# B&R Automation Studio project Nitto (part 13)

#### FB_Machine.st - TODO: Beinhaltet aller Baugrupen der Maschine
```iecst
(********************************************************************
 * COPYRIGHT -- Microsoft
 ********************************************************************
 * Library: UserSpilke
 * Datei: FB_Machine.st
 * Autor: Awalz
 * Erstellt: 24. März 2014
 ********************************************************************
 * Implementierung der Library UserSpilke
 ********************************************************************)

(* TODO: Beinhaltet aller Baugrupen der Maschine *)
FUNCTION_BLOCK FB_Machine

	ctrl(masterModul := masterModul,
		UnwinderUnit := UnwinderUnit,
		webbuffer := webbuffer,
		pullbreak := pullbreak ,
		cuttingunit1 := cuttingunit1,
		turngridwinder := turngridwinder,
		longcutter := longcutter,
		pullbreakSt := pullbreakSt,
		cuttingunit2 :=	cuttingunit2,
		catchbelt := catchbelt,
		conveyor := conveyor,
		webguidingbuffer := webguidingbuffer,
		webguiding := webguiding,
		emcy_inputs := emcy_inputs,summerystartstop := summerystartstop,
		IOs := IOs, panel := panel, safety := safety, gVarMachine := gVarMachine, switchcabinet := switchcabinet,
		packbelt := packbelt);  (**)

END_FUNCTION_BLOCK
```

#### FB_MachineIOs.st
```iecst
(********************************************************************
 * COPYRIGHT -- Microsoft
 ********************************************************************
 * Programm: MAIN
 * Datei: FB_MachineIOs.st
 * Autor: Awalz
 * Erstellt: 12. Mai 2014
 ********************************************************************
 * Implementierung des Programms MAIN
 ********************************************************************)

 (*<$Description$> TODO: Bitte Kommentar hier einzufügen </$Description$>*)
FUNCTION_BLOCK FB_MachineIOs
	ampel(clk := panel.clk);
	CEEPlug_o := CEEPlugON;
END_FUNCTION_BLOCK
```

#### Package Logical/MainMachineCtrl/MAIN/Mastermodul - Neues leeres Paket

#### FB_SpeedCtlrPid.st
```iecst
(********************************************************************
 * COPYRIGHT -- Microsoft
 ********************************************************************
 * Programm: MAIN
 * Datei: FB_SpeedCtlrPid.st
 * Autor: awalz
 * Erstellt: 10. Dezember 2014
 ********************************************************************
 * Implementierung des Programms MAIN
 ********************************************************************)

(* TODO: Bitte Kommentar hier einfügen *)
FUNCTION_BLOCK FB_SpeedCtlrPid
	IF firststart THEN
		LCRPIDpara_0.Kfbk			:= 2.0; // Anti-windup used
		LCRPIDpara_0.d_mode			:= LCRPID_D_MODE_E;	// differentiate control deviation
		LCRPIDpara_0.fbk_mode		:= LCRPID_FBK_MODE_INTERN;	// feedback of internal output
		LCRPID_0.mode				:= LCRPID_MODE_AUTO;	// Standard PID operating mod
		// 50.000 = 3 m/min
		LCRPID_0.Y_max				:= 10;	// percent
		LCRPID_0.Y_min				:= -10;// percent
		LCRPIDpara_0.invert			:= TRUE;
		LCRPIDpara_0.Kp				:= PID_Kp; //1.6; (*11*)//0.2//17.09.15 geändert
		LCRPIDpara_0.Tn				:= 7;// 6;	//(*1.1*)//7 //17.09.15 geändert
		LCRPIDpara_0.Tv				:= 0.0; // D-part
		LCRPIDpara_0.Tf				:= 0;(*0.020;*)
		LCRPIDpara_0.WX_max			:= 1000.0;
		LCRPIDpara_0.WX_min			:= -1000.0;
		LCRPID_0.ident				:= LCRPIDpara_0.ident;
		zeitkonstante				:= 0.1;
		lowPassEnable				:= TRUE;
		// Maximum controller output:
		firststart := FALSE;
	 END_IF
	lowPass.enable := lowPassEnable;
	IF dancepos >32767 THEN (* weil der Sensor zu nahe sitzt gibt es ein Ünerlauf*)
		test := 2000;
	ELSE
		test := dancepos;
	END_IF
	lowPass.x := INT_TO_REAL (test);
	lowPass.t := zeitkonstante; //2
	lowPass();
	lowPassSpeed.enable := TRUE;
	lowPassSpeed.x := INT_TO_REAL (ConveyerVelocity); // analog Input from conveyer
	lowPassSpeed.t := 3;
	lowPassSpeed();
//	lowPass.y_set := 0;
//	lowPass.set := TRUE;
//	rDancepos := INT_TO_REAL (dancepos) * SCALE_10V_TO_MM;
	rDancepos := lowPass.y * SCALE_10V_TO_MM; // gefilterte Tänzer position in mm
	inc_to_volt := lowPassSpeed.y * SCALE_INC_TO_V;
	volt_to_speed := maxMainVelocity /10 * inc_to_volt;

	LCRPIDpara_0();
	//************************** LCRPID *******************************
	LCRPID_0.ident						:= LCRPIDpara_0.ident;
	// PID controller:
	//  setpoint  		"W" = dancer position from application recipe
	//  actual value	"X" = measured act dancer position from analog input (*override wird beim füllen draufgegebe*)
	LCRPID_0.W			:= LIMIT (0, setDancerpos , 1000);
	LCRPID_0.X			:= rDancepos;  (*LCRPT1e_ActTension.y;*)
	LCRPID_0();
	(*OutPID				:= LCRPID_TM.Y * TM_SCALE_PID_OUT_TO_OFFSET;*)

	IF reset THEN
		setVelocity := LIMIT (0, volt_to_speed, 21); (*setVelocity;*) (*+ velocityOffset;*) (* Offset damit der Tänzer in der Mitte bleibt*) // OKrebs // statt 11 -> 21
	ELSE
		IF lowPassSpeed.y < 600 THEN //  weil das Signal drunter nur ein Rauschen ist
			tempvalue	:= 0;
		ELSE
			tempvalue		:= LIMIT (-3, LCRPID_0.Y * TM_SCALE_PID_OUT_TO_OFFSET, 3(*maxMainVelocity*)) ;
		END_IF
//		setVelocity := LIMIT (0,( volt_to_speed + tempvalue), 11); // OKrebs 12.04.17

		IF startCycleWebturrit THEN  // OKrebs // 12.04.17 // ANFANG
			IF NOT dancerWasEmpty THEN (*1*)
				setVelocity := LIMIT (0, volt_to_speed + 2, 21); // Geschwindigkeit erhöhen bis Tänzer leer ist // // OKrebs // statt 11 -> 21
			END_IF
			IF rDancepos < minDancerPos THEN  (*2*)// Wenn Tänzer leer/oben ist
				setVelocity := LIMIT (0, speedToCycleWebturrit, 21); // Geschwindigkeit verringern bis der Tänzer wieder voll ist // // OKrebs // statt 11 -> 21
				dancerWasEmpty := TRUE;
			END_IF
			IF dancerWasEmpty AND (rDancepos > maxDancerPos) THEN (*3*) // Wenn Tänzer wieder voll ist
				startCycleWebturrit := FALSE;
			END_IF
		ELSE
			setVelocity := LIMIT (0,( volt_to_speed + tempvalue), 21);  // // OKrebs // statt 11 -> 21
			dancerWasEmpty := FALSE;
		END_IF // OKrebs // ENDE

	END_IF
	// ================
	// CHECK ERRORS
	// ================

	IF (LCRPID_0.status > 12022) AND
	   (LCRPID_0.status < 65534) THEN
//		// Error in PID controller detected -> stop control
		AxisStep		:= ST_CTRL_OFF;
	END_IF

	CASE AxisStep OF
		//********************* INITIALISATION ************************
		ST_INIT1:
			LCRPIDpara_0.enable		:= TRUE;
			LCRPIDpara_0.enter		:= FALSE;
			LCRPID_0.enable			:= FALSE; (* 10.12.14*)
			AxisStep					:= ST_READY;

		//********************* WAIT FOR COMMANDS ************************
		ST_READY:
				LCRPID_0.enable			:= FALSE;
				AxisStep		:= ST_WAIT_POWER_ENABLED;
			// End of STEP_TM_READY
		//********************* WAIT FOR DRIVES BEING ENABLED ************************
		ST_WAIT_POWER_ENABLED:
		(*	IF  MC_ReadStatus_0.StandStill OR  MC_ReadStatus_0.ContinuousMotion THEN*)
				AxisStep			:= ST_LOAD_PARA_START;
				// Generate rising edge at the enter input in order to update
				// PID controller parameters
				LCRPIDpara_0.enter	:= FALSE;
			// End of STEP_TM_WAIT_POWER_ENABLED
		//********************* START PARAMETER LOADING ************************
		ST_LOAD_PARA_START:
			// Rising edge for updating controller parameter
			LCRPIDpara_0.enter		:= TRUE;
			AxisStep				:= ST_WAIT_LOAD_PARA_DONE;
//		//********************* WAIT FOR PARAMETER LOAD COMPLETE ************************
		ST_WAIT_LOAD_PARA_DONE:
			LCRPIDpara_0.enter		:= FALSE;
			AxisStep				:= ST_WAIT_SWITCH_CTRL_ON;
			// End of STEP_TM_WAIT_LOAD_PARA_DONE
//
//		//********************* ACTIVATE CONTROL ************************
		ST_WAIT_SWITCH_CTRL_ON:
			IF   (LCRPIDpara_0.ident <> 0)  THEN
				// Enable PID controller and Offset correction for web tension control
				LCRPID_0.enable				:= TRUE;
			(*	AxisStep						:= ST_CTRL_ACTIVE*);
			ELSIF reset THEN
				AxisStep := ST_INIT1;
			END_IF

	END_CASE

END_FUNCTION_BLOCK
```

#### FB_MASTERMODUL.st
```iecst
(********************************************************************
 * COPYRIGHT -- Microsoft
 ********************************************************************
 * Library: UserSpilke
 * Datei: FB_MASTERMODUL.st
 * Autor: Awalz
 * Erstellt: 25. März 2014
 ********************************************************************
 * Implementierung der Library UserSpilke
 ********************************************************************)

(*<$Description$> TODO: Bitte Kommentar hier einzufügen </$Description$>*)
FUNCTION_BLOCK FB_MASTERMODUL
END_FUNCTION_BLOCK
```

#### ac_automaticMaster.st
```iecst
(********************************************************************
 * COPYRIGHT -- Microsoft
 ********************************************************************
 * Programm: MAIN
 * Datei: ac_automaticMaster.st
 * Autor: Awalz
 * Erstellt: 1. April 2014
 ********************************************************************
 * Implementierung des Programms MAIN
 ********************************************************************)

 (*<$Description$> Fügt eine neue Aktion zum IEC Programm oder Bibliothek </$Description$>*)
ACTION ac_automaticMaster:
	CASE state OF
	ST_IDLE:
	(*	pulsHorn(IN := FALSE);*)

		IF BetrCtrl.value = CONST.MACHINEMODES.AUTOMATIC THEN
			handWheel.reset := TRUE;
			panel.LDTAutomatic.LDT.aktion := CONST.LAMP.BLINK500;
			panel.LDTJOG.LDT.aktion := CONST.LAMP.OFF;
		(*	errorKlemmungVornUnten.active := FALSE;
			errorKlemmungHintenUnten.active := FALSE;
			IF unitsStatus.durchmesserStop THEN
				errorDiameterStop.active := TRUE;
			ELSE
				errorDiameterStop.active := FALSE;
				IF unitsStatus.klemmungVornStop THEN
					errorKlemmungVornUnten.active := TRUE;
				ELSIF unitsStatus.klemmungHintenStop THEN
					errorKlemmungHintenUnten.active := TRUE;
				ELSIF unitsStatus.unwinderNotUp THEN
					errorUnwinderNotUp.active := TRUE;
				ELSE
					errorUnwinderNotUp.active := FALSE;*)
					IF unitsStatus.ready AND cuttingunit2.emcy_inputs.EMCY_DoorsClosed AND  cuttingunit1.emcy_inputs.EMCY_DoorsClosed AND  webbuffer.emcy_inputs.EMCY_DoorsClosed AND pullbreak.emcy_inputs.EMCY_DoorsClosed AND
				 longcutter.emcy_inputs.EMCY_DoorsClosed AND cuttingunit2.emcy_inputs.EMCY_DoorsClosed  AND safety.RequestSLS THEN
					(*AND unitsStatus.clampingback AND unitsStatus.clampingfront AND unitsStatus.clampingsplicetable *)
						(*NOT (UnwinderUnit.clamp.toDown_o OR UnwinderUnit.splicetable.clampAfter.toDown_o OR
						UnwinderUnit.splicetable.clampBefore.toDown_o OR UnwinderUnit.unwinderDrv.clamp.toDown_o
						OR UnwinderUnit.unwinderOp.clamp.toDown_o) THEN*)
						(*AND datacom.mach.loaded AND datacom.recipe.loaded AND datacom.tools.com.loaded THEN*)
						state := ST_AXIS_RUN;
					END_IF
				(*END_IF
			END_IF*)
		ELSE
			err(reset := TRUE);
			busy := TRUE;
			StateCtrl := CTRL_AUTO_AFTER;
		END_IF

	ST_AXIS_RUN:
		IF axis.busy OR axis.cmd <> CONST.AXIS.NOACTION THEN
			axis.cmd := CONST.AXIS.NOACTION;
		ELSE
			panel.LDTAutomatic.LDT.aktion := CONST.LAMP.ON;
			IOs.ampel.ondelay := T#3s;
			IOs.ampel.horn := TRUE;
			axis(cmd := CONST.AXIS.MOVE_VELOCITY, velocity := handWheel.setVelocity);
			state := ST_AXIS_RUN_FAST;
		END_IF
	(*	ELSE
			data.set.override := 0;
			axis.ctrl.ref.PlcToNc.Override := data.set.override;
			axis.ctrl( cmd := CONST.AXIS.START, position := axis.ctrl.ref.NcToPlc.ActPos + 9999999999999, velocity := STARTVELO);
			panels.autoLangsam.lamp.aktion :=  const.LAMP.BLINK500;
			panels.autoSchnell.lamp.aktion :=  const.LAMP.BLINK500;

			IOs.tasterflascheAbwickler.jog.lamp.aktion := const.LAMP.BLINK500;
			IOs.tasterflascheLongford.jog.lamp.aktion := const.LAMP.BLINK500;
			IOs.tasterflscheSpender.jog.lamp.aktion := const.LAMP.BLINK500;
			state := ST_AXIS_RUN_FAST;
		END_IF*)

	ST_AXIS_RUN_FAST:
		axis();
		IF  NOT safety.RequestSLS THEN
			IOs.ampel.Gelb.aktion := CONST.LAMP.BLINK500;
			panel.LDTRESET.LDT.aktion := CONST.LAMP.BLINK500; (* um zu signalisieren dass der Safetyrequest gedückt werden muss*)
		ELSE
			IOs.ampel.Gelb.aktion := CONST.LAMP.OFF;
			panel.LDTRESET.LDT.aktion := CONST.LAMP.OFF;
		END_IF
		 // Geschwindigkeitsänderung mit Handrad auf dem Panel
		axis(cmd := CONST.AXIS.MOVE_VELOCITY, velocity := handWheel.setVelocity);
		IF BetrCtrl.value = CONST.MACHINEMODES.MANUAL THEN
//			errorKlemmungVornUnten.active := FALSE;
//			errorKlemmungHintenUnten.active := FALSE;
//			errorDiameterStop.active := FALSE;
//			errorUnwinderNotUp.active := FALSE;
			axis(cmd := CONST.AXIS.STOP, ruck := 0, verzoegerung := 120000 );
			state := ST_AXIS_STOP;
		ELSIF BetrCtrl.value <> CONST.MACHINEMODES.AUTOMATIC OR NOT unitsStatus.ready OR NOT safety.RequestSLS  THEN
//			errorKlemmungVornUnten.active := FALSE;
//			errorKlemmungHintenUnten.active := FALSE;
//			errorDiameterStop.active := FALSE;
//			errorUnwinderNotUp.active := FALSE;
			axis( cmd := CONST.AXIS.STOP, ruck := 20000, verzoegerung := 120000 );
			state := ST_AXIS_STOP;
		ELSIF unitsStatus.diameterStop THEN
//		(*errorKlemmungVornUnten.active := FALSE;
//			errorKlemmungHintenUnten.active := FALSE;
//			errorUnwinderNotUp.active := FALSE;
//			errorDiameterStop.active := TRUE;*)
			axis( cmd := CONST.AXIS.STOP, ruck := 20000, verzoegerung := 120000);
			state := ST_AXIS_STOP;
//		ELSIF 	unitsStatus.clampingfront THEN
//			(*errorKlemmungVornUnten.active := TRUE;
//			errorKlemmungHintenUnten.active := FALSE;
//			errorUnwinderNotUp.active := FALSE;
//			errorDiameterStop.active := FALSE;*)
//			axis( cmd := CONST.AXIS.STOP, ruck := 20000, verzoegerung := 4000 );
//		(*	panels.stopSchnell.lamp.aktion := const.LAMP.ON; (*J.H.*)
//			state := ST_AXIS_STOP;
//		ELSIF unitsStatus.clampingback THEN
//		(*	errorKlemmungVornUnten.active := FALSE;
//			errorKlemmungHintenUnten.active := TRUE;
//			errorUnwinderNotUp.active := FALSE;
//			errorDiameterStop.active := FALSE;*)
//			axis( cmd := CONST.AXIS.STOP, ruck := 20000, verzoegerung := 4000 );
//			(*panels.stopSchnell.lamp.aktion := const.LAMP.ON; (*J.H.*)
//			state := ST_AXIS_STOP;
//		ELSIF unitsStatus.clampingsplicetable THEN
//		(*	errorKlemmungVornUnten.active := FALSE;
//			errorKlemmungHintenUnten.active := TRUE;
//			errorUnwinderNotUp.active := FALSE;
//			errorDiameterStop.active := FALSE;*)
//			axis( cmd := CONST.AXIS.STOP, ruck := 20000, verzoegerung := 4000 );
//			(*panels.stopSchnell.lamp.aktion := const.LAMP.ON; (*J.H.*)
//			state := ST_AXIS_STOP;
		END_IF

	ST_AXIS_VELO_CHANGE:
	(*	pulsHorn.IN := TRUE;
		axis.ctrl();
		timer();
		IF panels.runFast.key.rtrig.Q THEN
			IF data.set.override <> endOverride THEN
				data.set.override := endOverride;
			ELSE
				data.set.override := actOverride;
			END_IF
		END_IF*)
		IF BetrCtrl.value <> CONST.MACHINEMODES.AUTOMATIC OR NOT unitsStatus.ready THEN
			axis.verzoegerung :=120000;
			axis.cmd := CONST.AXIS.STOP;

			state := ST_AXIS_STOP;
	(*	ELSIF timer.Q THEN
			timer(in := FALSE);
			state := ST_AXIS_RUN_FAST;*)
		END_IF;

	ST_AXIS_STOP:

		IF NOT axis.busy THEN
			axis(cmd := CONST.AXIS.NOACTION);
			IF BetrCtrl.value <> CONST.MACHINEMODES.AUTOMATIC THEN
				busy := TRUE;
				panel.LDTAutomatic.LDT.aktion := CONST.LAMP.OFF;
				axis.cmd := CONST.AXIS.NOACTION;
				StateCtrl := CTRL_AUTO_AFTER;
			ELSE
				 IF NOT axis.busy THEN
					axis.cmd := CONST.AXIS.NOACTION;
					busy := FALSE;
					state := ST_IDLE;
				END_IF
			END_IF
		END_IF

//	ST_AXIS_UNWINDER_STOP:
//		axis.();
//		IF NOT axis.ctrl.Busy THEN
//			axis.ctrl(cmd := CONST.AXIS.NOACTION);
//			IF BetrCtrl.value <> CONST.MACHINEMODES.AUTOMATIC THEN
//				errorUnwinderNotUp.active := FALSE;
//				Busy := TRUE;
//				StateCtrl := CTRL_AUTO_AFTER;
//			ELSE
//				Busy := FALSE;
//			END_IF
//		END_IF*);

	ST_AXIS_DURCHMSTOP:

		IF NOT axis.busy THEN
			axis(cmd := CONST.AXIS.NOACTION);
			IF BetrCtrl.value <> CONST.MACHINEMODES.AUTOMATIC THEN
//				errorDiameterStop.active := FALSE;
				busy := TRUE;
				StateCtrl := CTRL_AUTO_AFTER;
			ELSE
				busy := FALSE;
			END_IF
		END_IF;

	ST_BAHN_END:
	(*	busy := FALSE;
		IF BetrCtrl.value <> CONST.MACHINEMODES.AUTOMATIC THEN
			state := ST_IDLE;
			err.reset();
			Busy := TRUE;
			StateCtrl := CTRL_AUTO_AFTER;
		END_IF*);

	ST_ERROR:
	(*	err.flag := TRUE;
		busy := FALSE;
		IF BetrCtrl.value <> CONST.MACHINEMODES.AUTOMATIC THEN
			state := ST_IDLE;
			err.reset();
			Busy := TRUE;
			StateCtrl := CTRL_AUTO_AFTER;
		END_IF*);
	END_CASE
END_ACTION
```

#### ac_manualMaster.st
```iecst
(********************************************************************
 * COPYRIGHT -- Microsoft
 ********************************************************************
 * Programm: MAIN
 * Datei: ac_manualMaster.st
 * Autor: Awalz
 * Erstellt: 1. April 2014
 ********************************************************************
 * Implementierung des Programms MAIN
 ********************************************************************)

 (*<$Description$> Fügt eine neue Aktion zum IEC Programm oder Bibliothek </$Description$>*)
ACTION ac_manualMaster:
		IF  NOT safety.RequestSLS THEN
			IOs.ampel.Gelb.aktion := CONST.LAMP.BLINK500;
			panel.LDTRESET.LDT.aktion := CONST.LAMP.BLINK500; (* um zu signalisieren dass der Safetyrequest gedückt werden muss*)
		ELSE
			IOs.ampel.Gelb.aktion := CONST.LAMP.OFF;
			panel.LDTRESET.LDT.aktion := CONST.LAMP.OFF;
		END_IF
	CASE state OF

	ST_IDLE:
		IF BetrCtrl.value = CONST.MACHINEMODES.MANUAL THEN
			axis.MC_ReadStatus_0();
			IF axis.MC_BR_ReadDriveStatus_0.Error THEN
				axis.cmd := CONST.AXIS.RESET;
				state := ST_RESET_WAIT;
			ELSIF unitsStatus.ready (*AND NOT (UnwinderUnit.clamp.toDown_o OR UnwinderUnit.splicetable.clampAfter.toDown_o OR
											 UnwinderUnit.splicetable.clampBefore.toDown_o OR UnwinderUnit.unwinderDrv.clamp.toDown_o
												OR UnwinderUnit.unwinderOp.clamp.toDown_o) *)THEN
				(*datacom.mach.loaded AND datacom.recipe.loaded AND datacom.tools.com.loaded*)
			(*	errorKlemmungVornUnten.active := FALSE;
				errorKlemmungHintenUnten.active := FALSE;
				panels.fwSlow.lamp.aktion := CONST.LAMP.BLINK500;*)
				panel.LDTJOG.LDT.aktion := CONST.LAMP.BLINK500;

				IF summerystartstop.jog AND safety.RequestSLS THEN (* alle Türen sind zu es darf von jeder Stelle gejoggt werden*)
					panel.LDTAutomatic.LDT.aktion := CONST.LAMP.OFF;
//					axis.BasicControl.Parameter.Acceleration := 5000;
//					axis.BasicControl.Parameter.Deceleration := 5000;
					axis(cmd := CONST.AXIS.JOG_POS, velocity := data.startSpeed/16666.67);
					panel.LDTJOG.LDT.aktion := CONST.LAMP.ON;
					busy := TRUE;
					state := ST_AXIS_RUN_SLOW;

				ELSIF cuttingunit1.emcy_inputs.EMCY_DoorsClosed AND webbuffer.emcy_inputs.EMCY_DoorsClosed AND longcutter.emcy_inputs.EMCY_DoorsClosed AND
					cuttingunit2.emcy_inputs.EMCY_DoorsClosed AND summerystartstop.boxwebbuffer.jog.LDT.button THEN
					axis(cmd := CONST.AXIS.JOG_POS, velocity := data.startSpeed/16666.67);
					panel.LDTJOG.LDT.aktion := CONST.LAMP.ON;
					busy := TRUE;
					state := ST_AXIS_RUN_SLOW_PB1;

				ELSIF  webbuffer.emcy_inputs.EMCY_DoorsClosed AND pullbreak.emcy_inputs.EMCY_DoorsClosed AND
				 longcutter.emcy_inputs.EMCY_DoorsClosed AND cuttingunit2.emcy_inputs.EMCY_DoorsClosed AND summerystartstop.boxcutting1.jog.LDT.button THEN
					axis(cmd := CONST.AXIS.JOG_POS, velocity := data.startSpeed/16666.67);
					panel.LDTJOG.LDT.aktion := CONST.LAMP.ON;
					busy := TRUE;
					state := ST_AXIS_RUN_SLOW_CUT1;
				ELSIF webbuffer.emcy_inputs.EMCY_DoorsClosed AND pullbreak.emcy_inputs.EMCY_DoorsClosed AND cuttingunit1.emcy_inputs.EMCY_DoorsClosed AND
					summerystartstop.boxlongcutter.jog.LDT.button THEN
					axis(cmd := CONST.AXIS.JOG_POS, velocity := data.startSpeed/16666.67);
					panel.LDTJOG.LDT.aktion := CONST.LAMP.ON;
					busy := TRUE;
					state := ST_AXIS_RUN_SLOW_CUT2;
				END_IF

			ELSE
				IF unitsStatus.clampingfront  THEN
					errorclampingfront.active := TRUE;
				ELSE
					errorclampingfront.active := FALSE;
				END_IF
				IF unitsStatus.clampingback THEN
					errorclampingback.active := TRUE;
				ELSE
					errorclampingback.active := FALSE;
				END_IF
			END_IF
		ELSE
			axis(cmd := CONST.AXIS.NOACTION);
			busy := TRUE;
			StateCtrl := CTRL_MANUAL_AFTER;
		END_IF

	ST_AXIS_RUN_SLOW:
		axis();
		IF BetrCtrl.value <> CONST.MACHINEMODES.MANUAL OR NOT unitsStatus.ready OR NOT summerystartstop.jog  THEN
			axis.MC_ReadStatus_0();
			axis.verzoegerung := 120000;
			axis(cmd := CONST.AXIS.STOP);
			state := ST_AXIS_STOP;
		END_IF

//
	ST_AXIS_RUN_SLOW_PB1:
			axis();
		IF BetrCtrl.value <> CONST.MACHINEMODES.MANUAL OR NOT unitsStatus.ready OR NOT summerystartstop.			boxwebbuffer.jog.LDT.button OR NOT webbuffer.emcy_inputs.EMCY_DoorsClosed
		OR NOT cuttingunit1.emcy_inputs.EMCY_DoorsClosed OR NOT longcutter.emcy_inputs.EMCY_DoorsClosed 			OR NOT cuttingunit2.emcy_inputs.EMCY_DoorsClosed THEN
			axis.MC_ReadStatus_0();
			axis.verzoegerung := 120000;
			axis(cmd := CONST.AXIS.STOP);
			state := ST_AXIS_STOP;
		END_IF

	ST_AXIS_RUN_SLOW_CUT1:
			axis();
		IF BetrCtrl.value <> CONST.MACHINEMODES.MANUAL OR NOT unitsStatus.ready OR NOT summerystartstop.			boxcutting1.jog.LDT.button OR NOT webbuffer.emcy_inputs.EMCY_DoorsClosed
		OR NOT pullbreak.emcy_inputs.EMCY_DoorsClosed OR NOT longcutter.emcy_inputs.EMCY_DoorsClosed OR 			NOT cuttingunit2.emcy_inputs.EMCY_DoorsClosed THEN
			axis.MC_ReadStatus_0();
			axis.verzoegerung := 80000;
			axis(cmd := CONST.AXIS.STOP);
			state := ST_AXIS_STOP;
		END_IF

	ST_AXIS_RUN_SLOW_CUT2:
			axis();
		IF BetrCtrl.value <> CONST.MACHINEMODES.MANUAL OR NOT unitsStatus.ready OR NOT summerystartstop.			boxlongcutter.jog.LDT.button OR NOT webbuffer.emcy_inputs.EMCY_DoorsClosed
		OR NOT pullbreak.emcy_inputs.EMCY_DoorsClosed  OR NOT cuttingunit1.emcy_inputs.EMCY_DoorsClosed 		THEN
			axis.MC_ReadStatus_0();
			axis.verzoegerung := 120000;
			axis(cmd := CONST.AXIS.STOP);
			state := ST_AXIS_STOP;
		END_IF

	ST_AXIS_STOP:
		IF NOT axis.busy THEN
			axis(cmd := CONST.AXIS.NOACTION);
			IF BetrCtrl.value <> CONST.MACHINEMODES.MANUAL THEN
				busy := TRUE;
				StateCtrl := CTRL_MANUAL_AFTER;
			ELSE
				busy := FALSE;
			END_IF
			state := ST_IDLE;
		END_IF

	ST_RESET_WAIT:
		axis();
		IF NOT axis.busy THEN
			axis.cmd := CONST.AXIS.NOACTION;
			state := ST_IDLE;
		END_IF

	ST_ERROR:
		busy := FALSE;
		IF BetrCtrl.value <> CONST.MACHINEMODES.MANUAL THEN
			state := ST_IDLE;
			(*err.reset();*)
			busy := TRUE;
			StateCtrl := CTRL_MANUAL_AFTER;
		END_IF;

	END_CASE

END_ACTION
```

#### ac_setStateAfterMaster.st
```iecst
(********************************************************************
 * COPYRIGHT -- Microsoft
 ********************************************************************
 * Programm: MAIN
 * Datei: ac_setStateAfterMaster.st
 * Autor: Awalz
 * Erstellt: 1. April 2014
 ********************************************************************
 * Implementierung des Programms MAIN
 ********************************************************************)

 (*<$Description$> Fügt eine neue Aktion zum IEC Programm oder Bibliothek </$Description$>*)
ACTION ac_setStateAfterMaster:
	IF BetrCtrl.value = CONST.MACHINEMODES.EMERGENCYSTOP THEN
		StateCtrl := CTRL_EMERGENCYSTOP_BEFORE;
	ELSIF BetrCtrl.value = CONST.MACHINEMODES.SAFETYSTOP THEN
		StateCtrl := CTRL_SAFETYSTOP_BEFORE;
	ELSIF BetrCtrl.value = CONST.MACHINEMODES.MANUAL THEN
		StateCtrl := CTRL_STOP;
	ELSIF BetrCtrl.value = CONST.MACHINEMODES.AUTOMATIC THEN
		StateCtrl := CTRL_STOP;
	END_IF

END_ACTION
```

#### ac_inline.st
```iecst
(********************************************************************
 * COPYRIGHT -- Microsoft
 ********************************************************************
 * Programm: MAIN
 * Datei: ac_inline.st
 * Autor: awalz
 * Erstellt: 22. August 2014
 ********************************************************************
 * Implementierung des Programms MAIN
 ********************************************************************)

(* Fügt eine neue Aktion zum IEC Programm oder Bibliothek *)
ACTION ac_inline:
CASE state OF
	ST_IDLE:

		IF BetrCtrl.value = CONST.MACHINEMODES.AUTOMATIC THEN
			IF unitsStatus.ready (*AND unitsStatus.clampingback AND unitsStatus.clampingfront AND unitsStatus.clampingsplicetable *)THEN
						state := ST_AXIS_RUN;
			END_IF

		ELSE
			err(reset := TRUE);
			busy := TRUE;
			StateCtrl := CTRL_AUTO_AFTER;
		END_IF

	ST_AXIS_RUN:
		IF axis.busy OR axis.cmd <> CONST.AXIS.NOACTION THEN
			axis.cmd := CONST.AXIS.NOACTION;
		ELSE
			panel.LDTAutomatic.LDT.aktion := CONST.LAMP.ON;
			IOs.ampel.ondelay := T#5s;
			IOs.ampel.horn := TRUE;
			axis(cmd := CONST.AXIS.MOVE_VELOCITY, velocity := inlineVelocity.setVelocity);
			IOs.machineReady := TRUE;
			state := ST_AXIS_RUN_FAST;
		END_IF

	ST_AXIS_RUN_FAST:
	(*	axis();	*)
		IF  NOT safety.RequestSLS THEN (*gelbe Ampel blinken lassen wenn die Safety speed nicht freigegeben ist*)
			IOs.ampel.Gelb.aktion := CONST.LAMP.BLINK500;
			panel.LDTRESET.LDT.aktion := CONST.LAMP.BLINK500;
		ELSE
			IOs.ampel.Gelb.aktion := CONST.LAMP.OFF;
				panel.LDTRESET.LDT.aktion := CONST.LAMP.OFF;

		END_IF
 		// Geschwindigkeitsänderung abhängig vom Tänzer des Zufuhr
		axis(cmd := CONST.AXIS.MOVE_VELOCITY, velocity := inlineVelocity.setVelocity);
		IF BetrCtrl.value = CONST.MACHINEMODES.MANUAL THEN
			axis(cmd := CONST.AXIS.STOP, ruck := 2000, verzoegerung := 40000 );
			state := ST_AXIS_STOP;
		ELSIF BetrCtrl.value <> CONST.MACHINEMODES.AUTOMATIC OR NOT unitsStatus.ready OR NOT safety.RequestSLS THEN
			axis( cmd := CONST.AXIS.STOP, ruck := 20000, verzoegerung := 80000 );
			state := ST_AXIS_STOP;
		END_IF

	ST_AXIS_STOP:
		IF  NOT axis.busy THEN
			axis(cmd := CONST.AXIS.NOACTION);
			IF BetrCtrl.value <> CONST.MACHINEMODES.AUTOMATIC THEN
				busy := TRUE;
				IOs.machineReady := FALSE;
				panel.LDTAutomatic.LDT.aktion := CONST.LAMP.OFF;
				axis.cmd := CONST.AXIS.NOACTION;
				StateCtrl := CTRL_AUTO_AFTER;
			ELSE
			 	IF NOT axis.busy THEN
					axis.cmd := CONST.AXIS.NOACTION;
					busy := FALSE;
					state := ST_IDLE;
				END_IF
			END_IF
		END_IF

	ST_ERROR:
	err.flag := TRUE;
		busy := FALSE;
		IF BetrCtrl.value <> CONST.MACHINEMODES.AUTOMATIC THEN
			state := ST_IDLE;
			err(reset := TRUE);
			busy := TRUE;
			StateCtrl := CTRL_AUTO_AFTER;
		END_IF;
	END_CASE
END_ACTION
```

#### FB_MasterModulCtrl.st
```iecst
(********************************************************************
 * COPYRIGHT -- Microsoft
 ********************************************************************
 * Library: UserSpilke
 * Datei: FB_MasterModulCtrl.st
 * Autor: Awalz
 * Erstellt: 25. März 2014
 ********************************************************************
 * Implementierung der Library UserSpilke
 ********************************************************************)

(*<$Description$> Hier wird die MasterAchse in Bewegung gesetzt da die andere Module gekoppelt sind führen diese die gleiche Bewegung aus </$Description$>*)
FUNCTION_BLOCK FB_MasterModulCtrl
	unitsStatus( UnwinderUnit := UnwinderUnit, pullbreak := pullbreak, pullbreakSt := pullbreakSt,
				conveyor := conveyor, catchbelt := catchbelt, longcutter := longcutter, cuttingunit1 := cuttingunit1, cuttingunit2 := cuttingunit2, webbuffer := webbuffer, turngridwinder := turngridwinder); // OKrebs 09.12.15
	axis();
	IOs(panel := panel);
	safety();
	sprayCtrl(machineaxis := axis, length1 := data.lenght1, length2 := data.lenght2);
	IF buttonSprayVisu THEN
		sprayCtrl.valveout := TRUE;
	END_IF
	summerystartstop(clk := panel.clk, panel := panel);
	axis.BasicControl.Parameter.Deceleration	:= 80000.0; //only for initialization
	axis.BasicControl.Parameter.Acceleration	:= 80000.0;
//	axis.MC_ReadActualVelocity_0();
//	mastervelocity := axis.MC_ReadActualVelocity_0.Velocity;
	//	handWheel( actualVelocity := mastervelocity, limitspeed := data.maxSpeed, safetyspeedrequest := safety.RequestSLS);
	handWheel( actualVelocity := axis.MC_ReadActualVelocity_0.Velocity, limitspeed := data.maxSpeed, safetyspeedrequest := safety.RequestSLS);
	inlineVelocity( limitspeed := 0, setDancerpos := 500, maxMainVelocity := 20, speedToCycleWebturrit := data.speedToCycleWebturrit/16666.67); //OKrebs //28.06.17 // vorher maxMainVelocity := 10

CASE StateCtrl OF
    CTRL_FIRST_START:
		busy := TRUE;
		StateCtrl := CTRL_EMERGENCYSTOP_BEFORE;

	CTRL_MANUAL_BEFORE:
		axis.BasicControl.Command.Power := TRUE;
		IF BetrCtrl.value = CONST.MACHINEMODES.MANUAL THEN
			(*BetrStatus.set := TRUE;*)
			BetrStatus(set := TRUE, value := BetrCtrl.value);
			err(reset := TRUE);
		(*	axis.ctrl.setOverride();
			axis.ctrl.ref.PlcToNc.Override := 1000000;
			err.reset();*)
			busy := FALSE;
			state := ST_IDLE;
			IOs.ampel.Gelb.aktion := CONST.LAMP.OFF;
			panel.LDTRESET.LDT.aktion := CONST.LAMP.OFF;
			panel.LDTAutomatic.LDT.aktion := CONST.LAMP.OFF;
			StateCtrl := CTRL_MANUAL;
		ELSIF BetrCtrl.value = CONST.MACHINEMODES.EMERGENCYSTOP THEN
			StateCtrl := CTRL_EMERGENCYSTOP_BEFORE;
		ELSIF BetrCtrl.value = CONST.MACHINEMODES.SAFETYSTOP THEN
			StateCtrl := CTRL_SAFETYSTOP_BEFORE;
		ELSIF BetrCtrl.value = CONST.MACHINEMODES.AUTOMATIC THEN
			StateCtrl := CTRL_AUTO_BEFORE;
		END_IF

	CTRL_MANUAL:
		err(reset := FALSE);
		ac_manualMaster;

	CTRL_MANUAL_AFTER:
		ac_setStateAfterMaster;

	CTRL_AUTO_BEFORE:
		IF BetrCtrl.value = CONST.MACHINEMODES.AUTOMATIC THEN
			BetrStatus(set := TRUE, value := BetrCtrl.value);
			err(reset := TRUE);
			busy := FALSE;
			state := ST_IDLE;
		(*	axis.ctrl.setOverride();*)
//			IF data.recipe.startSpeed < 0.01 THEN
//				tmpStartOverride :=	(1*1000/60) / STARTVELO;
//			ELSIF data.recipe.startSpeed > 20 THEN
//				tmpStartOverride :=	(20*1000/60) / STARTVELO;
//			ELSE
//				tmpStartOverride :=	(data.recipe.startSpeed*1000/60) / STARTVELO;
//			END_IF
//			startOverride := LREAL_TO_UDINT(tmpStartOverride * 1000000);
//
//			IF data.recipe.startSpeed > data.recipe.maxSpeed THEN
//				tmpEndOverride :=	(data.recipe.startSpeed*1000/60) / STARTVELO;
//(* 30 ist zu viel, geändert J.H. 31.01.11
//			IF data.recipe.maxSpeed < 30 THEN
//				tmpEndOverride :=	(30*1000/60) / STARTVELO;
//*)			ELSIF data.recipe.maxSpeed > 180 THEN
//				tmpEndOverride :=	(180*1000/60) / STARTVELO;
//			ELSE
//				tmpEndOverride :=	(data.recipe.maxSpeed*1000/60) / STARTVELO;
//			END_IF

			StateCtrl := CTRL_AUTO;
		axis.BasicControl.Command.Power := TRUE;
		BetrStatus(set := TRUE, value := CONST.MACHINEMODES.EMERGENCYSTOP);
			StateCtrl := CTRL_AUTO;
		ELSIF BetrCtrl.value = CONST.MACHINEMODES.EMERGENCYSTOP THEN
			StateCtrl := CTRL_EMERGENCYSTOP_BEFORE;
		ELSIF BetrCtrl.value = CONST.MACHINEMODES.SAFETYSTOP THEN
			StateCtrl := CTRL_SAFETYSTOP_BEFORE;
		ELSIF BetrCtrl.value = CONST.MACHINEMODES.MANUAL THEN
			StateCtrl := CTRL_MANUAL_BEFORE;
		END_IF

	CTRL_AUTO:
		IF NOT IOs.inline AND NOT mainconvoyerrun THEN
			ac_automaticMaster;
		ELSIF IOs.inline(* inline AND mainconvoyerrun*) THEN
			ac_inline;
		END_IF

	CTRL_AUTO_AFTER:
		ac_setStateAfterMaster;
		panel.LDTAutomatic.LDT.aktion := CONST.LAMP.BLINK500;

	CTRL_STOP:
		IF BetrCtrl.value = CONST.MACHINEMODES.EMERGENCYSTOP THEN
			StateCtrl := CTRL_EMERGENCYSTOP_BEFORE;
		ELSIF BetrCtrl.value = CONST.MACHINEMODES.SAFETYSTOP THEN
			StateCtrl := CTRL_SAFETYSTOP_BEFORE;
		ELSE
			state := ST_IDLE;
			StateCtrl := CTRL_STOP_AFTER;
		END_IF

	CTRL_STOP_AFTER:
		IF BetrCtrl.value = CONST.MACHINEMODES.EMERGENCYSTOP THEN
			StateCtrl := CTRL_EMERGENCYSTOP_BEFORE;
		ELSIF BetrCtrl.value = CONST.MACHINEMODES.SAFETYSTOP THEN
			StateCtrl := CTRL_SAFETYSTOP_BEFORE;
		ELSIF BetrCtrl.value = CONST.MACHINEMODES.MANUAL THEN
			StateCtrl := CTRL_MANUAL_BEFORE;
		ELSIF BetrCtrl.value = CONST.MACHINEMODES.AUTOMATIC THEN
			StateCtrl := CTRL_AUTO_BEFORE;
		END_IF

	CTRL_RESET_START:
		BetrStatus (set := TRUE, value := CONST.MACHINEMODES.RESET);
		IF BetrCtrl.value = CONST.MACHINEMODES.EMERGENCYSTOP THEN
			StateCtrl := CTRL_EMERGENCYSTOP_BEFORE;
		ELSIF BetrCtrl.value = CONST.MACHINEMODES.SAFETYSTOP THEN
			StateCtrl := CTRL_SAFETYSTOP_BEFORE;
		ELSE
			StateCtrl := CTRL_RESET;
		END_IF

	CTRL_RESET:
		IF BetrCtrl.value = CONST.MACHINEMODES.EMERGENCYSTOP THEN
			StateCtrl := CTRL_EMERGENCYSTOP_BEFORE;
		ELSIF BetrCtrl.value = CONST.MACHINEMODES.SAFETYSTOP THEN
			StateCtrl := CTRL_SAFETYSTOP_BEFORE;
		ELSE
			StateCtrl := CTRL_RESET_AFTER;
		END_IF

	CTRL_RESET_AFTER:
		IF BetrCtrl.value = CONST.MACHINEMODES.RESET THEN
			busy := FALSE;
		ELSE
			busy := TRUE;
			err(reset := FALSE);
			IF BetrCtrl.value = CONST.MACHINEMODES.EMERGENCYSTOP THEN
				StateCtrl := CTRL_EMERGENCYSTOP_BEFORE;
			ELSIF BetrCtrl.value = CONST.MACHINEMODES.SAFETYSTOP THEN
				StateCtrl := CTRL_SAFETYSTOP_BEFORE;
			ELSIF BetrCtrl.value = CONST.MACHINEMODES.MANUAL THEN
				axis.cmd := CONST.AXIS.POWER_ON; (* Regler EInschalten *)
				StateCtrl := CTRL_MANUAL_BEFORE;
			ELSIF BetrCtrl.value = CONST.MACHINEMODES.AUTOMATIC THEN
				axis.cmd := CONST.AXIS.POWER_ON; (* Regler EInschalten *)
				StateCtrl := CTRL_AUTO_BEFORE;
			END_IF
		END_IF
(****neu 30.04***)
	CTRL_SAFETYSTOP_BEFORE:			(* Runter Rampen *)
		IF BetrCtrl.value = CONST.MACHINEMODES.EMERGENCYSTOP THEN
			StateCtrl := CTRL_EMERGENCYSTOP_BEFORE;
		ELSE
			axis.verzoegerung:= CONST.AXIS.EMERGENCY_DECELERATION; (* von 200m/min in 3 sek*)
			axis.cmd := CONST.AXIS.STOP;
			state := ST_IDLE;
			StateCtrl := CTRL_SAFETYSTOP;
		END_IF

	CTRL_SAFETYSTOP:
		IF BetrCtrl.value = CONST.MACHINEMODES.EMERGENCYSTOP THEN
			StateCtrl := CTRL_EMERGENCYSTOP_BEFORE;
		ELSE
//			CASE state OF
//			ST_IDLE:
//				IF axis.BasicControl.AxisState.StandStill OR axis.BasicControl.AxisState.StandStill  THEN
//
//					state := ST_QUIT;
//				END_IF
//
//			ST_QUIT:
//				state := ST_QUIT;
//				BetrStatus(set := TRUE,value := CONST.MACHINEMODES.SAFETYSTOP);
//				StateCtrl := CTRL_SAFETYSTOP_AFTER;
				//			END_CASE
			BetrStatus(set := TRUE,value := CONST.MACHINEMODES.SAFETYSTOP);
			IF axis.MC_ReadStatus_0.StandStill THEN
				axis.cmd := CONST.AXIS.NOACTION;//da virtuelle Achse
				StateCtrl := CTRL_SAFETYSTOP_AFTER;
			END_IF
		END_IF

	CTRL_SAFETYSTOP_AFTER:
		busy := FALSE;
		(*axis(cmd := CONST.AXIS.VAXIS_ON);*)
		IF BetrCtrl.value = CONST.MACHINEMODES.EMERGENCYSTOP THEN
			busy := TRUE;
			StateCtrl := CTRL_EMERGENCYSTOP_BEFORE;
		ELSIF BetrCtrl.value = CONST.MACHINEMODES.MANUAL THEN
			busy := TRUE;
			StateCtrl := CTRL_MANUAL_BEFORE;
		ELSIF BetrCtrl.value = CONST.MACHINEMODES.AUTOMATIC THEN
			busy := TRUE;
			StateCtrl := CTRL_AUTO_BEFORE;
		END_IF
(******)

	CTRL_EMERGENCYSTOP_BEFORE:
		BetrStatus(set := TRUE, value := CONST.MACHINEMODES.EMERGENCYSTOP);
		IF  axis.MC_ReadStatus_0.ContinuousMotion OR axis.MC_ReadStatus_0.DiscreteMotion
			OR axis.MC_ReadStatus_0.SynchronizedMotion  THEN
			axis.verzoegerung:= CONST.AXIS.EMERGENCY_DECELERATION;// 1111111;//11.03.15 1111111; (*200m/min = 3333334/3 in 3 sek*)
			axis.cmd := CONST.AXIS.STOP;
			state := ST_IDLE;
			StateCtrl := CTRL_EMERGENCYSTOP;
		ELSE //wenn die Maschine eingeschaltet wird
			axis.cmd := CONST.AXIS.NOACTION;
			state := ST_IDLE;
			StateCtrl := CTRL_EMERGENCYSTOP;
		END_IF

		CTRL_EMERGENCYSTOP:
		panel.LDTAutomatic.LDT.aktion :=  CONST.LAMP.OFF;
		IF BetrCtrl.value = CONST.MACHINEMODES.EMERGENCYSTOP THEN
			IF axis.MC_ReadStatus_0.StandStill THEN
				axis.cmd := CONST.AXIS.NOACTION;//da bei B&R eine virtulle Achse nicht ausgeschalten werden kann
				busy := FALSE;
			ELSIF axis.MC_ReadStatus_0.Disabled THEN
				axis.cmd := CONST.AXIS.NOACTION;
				busy := FALSE;
			END_IF
		ELSE
			err.reset := TRUE;
			busy := TRUE;
			StateCtrl := CTRL_RESET_START;
		END_IF
END_CASE

END_FUNCTION_BLOCK
```

#### Package Logical/MainMachineCtrl/MAIN/MainUnwinding - Neues leeres Paket

#### FB_MainUnwinder.st - TODO: Daten FB für Abwickler 
```iecst
(********************************************************************
 * COPYRIGHT -- Microsoft
 ********************************************************************
 * Library: UserSpilke
 * Datei: FB_MainUnwinder.st
 * Autor: Awalz
 * Erstellt: 24. März 2014
 ********************************************************************
 * Implementierung der Library UserSpilke
 ********************************************************************)

(* TODO: Daten FB für Abwickler  *)
FUNCTION_BLOCK FB_UNWINDER
//	IF data.recipeData.mode = 2 THEN
//		Push_Button_Mode_Led := TRUE;
//	ELSE
//		Push_Button_Mode_Led := FALSE;
//	END_IF

//	UnwinderModeTrig(CLK :=Push_Button_Mode );

//	IF UnwinderModeTrig.Q = TRUE AND data.recipeData.mode = 2 THEN
//		data.recipeData.mode := 1;
//	ELSE
//		IF UnwinderModeTrig.Q = TRUE AND data.recipeData.mode = 1 THEN
//			data.recipeData.mode :=2;
//		ELSE
//		END_IF
//	END_IF

END_FUNCTION_BLOCK
```

#### ac_manualUnwinder.st
```iecst
(********************************************************************
 * COPYRIGHT -- Microsoft
 ********************************************************************
 * Programm: MAIN
 * Datei: ac_manualUnwinder.st
 * Autor: Awalz
 * Erstellt: 7. April 2014
 ********************************************************************
 * Implementierung des Programms MAIN
 ********************************************************************)

 (*<$Description$> Fügt eine neue Aktion zum IEC Programm oder Bibliothek </$Description$>*)
ACTION ac_manualUnwinder:
		(*gehört zu MainUnwinderCtrl*)
		CASE state OF
	ST_IDLE:
		IF BetrCtrl.value <> CONST.MACHINEMODES.MANUAL THEN
			state := ST_IDLE;
			err(reset := TRUE);
			busy := TRUE;
		(*	status.ready := FALSE;*)
			StateCtrl := CTRL_MANUAL_AFTER;
		ELSE
			IF NOT feederCtrl.LimitSwitchRight AND machineaxis.MC_ReadStatus_0.ContinuousMotion THEN
				unwinderOp.data.recipeData.mode := CONST.UNITMODEs.ENABLE;
				state := ST_AXIS_RUN;	(*automatische aktivierung des Wicklers der gerade dran ist*)
			ELSIF NOT feederCtrl.LimitSwitchLeft AND  machineaxis.MC_ReadStatus_0.ContinuousMotion THEN
				unwinderDrv.data.recipeData.mode := CONST.UNITMODEs.ENABLE;
				state := ST_AXIS_RUN; (*automatische aktivierung des Wicklers der gerade dran ist*)
			ELSIF NOT feederCtrl.LimitSwitchRight AND  unwinderDrv.data.recipeData.mode = CONST.UNITMODEs.ENABLE THEN
				unwinderDrv.data.recipeData.mode := CONST.UNITMODEs.AXIS_OFF;
				state := ST_AXIS_STOP;(*automatische deaktivierung des Wicklers der gerade nicht dran ist*)
			ELSIF NOT feederCtrl.LimitSwitchLeft AND  unwinderOp.data.recipeData.mode = CONST.UNITMODEs.ENABLE THEN
				unwinderOp.data.recipeData.mode := CONST.UNITMODEs.AXIS_OFF;
				state := ST_AXIS_STOP;	(*automatische deaktivierung des Wicklers der gerade nicht dran ist*)
			END_IF
		END_IF

		ST_AXIS_RUN:
			IF BetrCtrl.value <> CONST.MACHINEMODES.MANUAL THEN
				state := ST_IDLE;
				err(reset := TRUE);
				busy := TRUE;
			(*	status.ready := FALSE;*)
				StateCtrl := CTRL_MANUAL_AFTER;
			ELSE
				IF NOT  machineaxis.MC_ReadStatus_0.ContinuousMotion THEN
					state := ST_IDLE;
				END_IF
			END_IF

		ST_AXIS_STOP:
			IF BetrCtrl.value <> CONST.MACHINEMODES.MANUAL THEN
				state := ST_IDLE;
				err(reset := TRUE);
				busy := TRUE;
			(*	status.ready := FALSE;*)
				StateCtrl := CTRL_MANUAL_AFTER;
			ELSE
				IF NOT  machineaxis.MC_ReadStatus_0.StandStill THEN
					state := ST_IDLE;
				END_IF
			END_IF
	END_CASE
END_ACTION
```

#### ac_automUnwinder.st
```iecst
(********************************************************************
 * COPYRIGHT -- Microsoft
 ********************************************************************
 * Programm: MAIN
 * Datei: ac_automUnwinder.st
 * Autor: awalz
 * Erstellt: 24. Juli 2014
 ********************************************************************
 * Implementierung des Programms MAIN
 ********************************************************************)

(* Fügt eine neue Aktion zum IEC Programm oder Bibliothek *)
ACTION ac_automUnwinder:
	CASE state OF
		ST_IDLE:
			IF BetrCtrl.value <> CONST.MACHINEMODES.AUTOMATIC  THEN
				state := ST_IDLE;
				err(reset := TRUE);
				busy := TRUE;
				(*	status.ready := FALSE;*)
				StateCtrl := CTRL_AUTO_AFTER;
			ELSE
				IF NOT feederCtrl.LimitSwitchRight AND machineaxis.MC_ReadStatus_0.ContinuousMotion THEN
					unwinderOp.data.recipeData.mode := CONST.UNITMODEs.ENABLE;
					state := ST_AXIS_RUN;
				ELSIF NOT feederCtrl.LimitSwitchLeft AND  machineaxis.MC_ReadStatus_0.ContinuousMotion THEN
					unwinderDrv.data.recipeData.mode := CONST.UNITMODEs.ENABLE;
					state := ST_AXIS_RUN;
				ELSIF NOT feederCtrl.LimitSwitchRight AND  unwinderDrv.data.recipeData.mode = CONST.UNITMODEs.ENABLE THEN
					unwinderDrv.data.recipeData.mode := CONST.UNITMODEs.AXIS_OFF;
					state := ST_AXIS_STOP; (*automatische deaktivierung des Wicklers der gerade nicht dran ist*)
				ELSIF NOT feederCtrl.LimitSwitchLeft AND unwinderOp.data.recipeData.mode = CONST.UNITMODEs.ENABLE THEN
					unwinderOp.data.recipeData.mode := CONST.UNITMODEs.AXIS_OFF;
					state := ST_AXIS_STOP;	(*automatische deaktivierung des Wicklers der gerade nicht dran ist*)
				END_IF
			END_IF

		ST_AXIS_RUN:
			IF BetrCtrl.value <> CONST.MACHINEMODES.AUTOMATIC THEN
				state := ST_IDLE;
				err(reset := TRUE);
				busy := TRUE;
				(*	status.ready := FALSE;*)
				StateCtrl := CTRL_AUTO_AFTER;
			ELSE
				IF NOT  machineaxis.MC_ReadStatus_0.ContinuousMotion (*AND NOT unwinderaxis.MC_ReadStatus_0.StandStill *) THEN
					state := ST_IDLE;
				END_IF
			END_IF

		ST_AXIS_STOP:
			IF BetrCtrl.value <> CONST.MACHINEMODES.AUTOMATIC THEN
				state := ST_IDLE;
				err(reset := TRUE);
				busy := TRUE;
				(*	status.ready := FALSE;*)
				StateCtrl := CTRL_AUTO_AFTER;
			ELSE
				IF NOT  machineaxis.MC_ReadStatus_0.StandStill (*AND NOT unwinderaxis.MC_ReadStatus_0.StandStill *) THEN
					state := ST_IDLE;
				END_IF
			END_IF
	END_CASE
END_ACTION
```

#### ac_setStateAfterUnwinder.st
```iecst
(********************************************************************
 * COPYRIGHT -- Microsoft
 ********************************************************************
 * Programm: MAIN
 * Datei: ac_setStateAfterUnwinder.st
 * Autor: Awalz
 * Erstellt: 7. April 2014
 ********************************************************************
 * Implementierung des Programms MAIN
 ********************************************************************)

 (*<$Description$> Fügt eine neue Aktion zum IEC Programm oder Bibliothek </$Description$>*)
ACTION ac_setStateAfterUnwinder:
	IF BetrCtrl.value = CONST.MACHINEMODES.EMERGENCYSTOP THEN
		StateCtrl := CTRL_EMERGENCYSTOP_BEFORE;
	ELSIF BetrCtrl.value = CONST.MACHINEMODES.SAFETYSTOP THEN
		StateCtrl := CTRL_SAFETYSTOP_BEFORE;
	ELSIF BetrCtrl.value = CONST.MACHINEMODES.MANUAL THEN
		StateCtrl := CTRL_STOP_BEFORE;
	ELSIF BetrCtrl.value = CONST.MACHINEMODES.AUTOMATIC THEN
		StateCtrl := CTRL_STOP_BEFORE;
	END_IF
END_ACTION
```

#### FB_UNWINDERUNIT.st
```iecst
(********************************************************************
 * COPYRIGHT -- Microsoft
 ********************************************************************
 * Programm: MAIN
 * Datei: FB_UNWINDERUNIT.st
 * Autor: Awalz
 * Erstellt: 23. Juni 2014
 ********************************************************************
 * Implementierung des Programms MAIN
 ********************************************************************)

(* TODO: Bitte Kommentar hier einfügen *)
FUNCTION_BLOCK FB_UNWINDERUNIT
END_FUNCTION_BLOCK
```

#### FB_MainUnwinderCtrl.st
```iecst
(********************************************************************
 * COPYRIGHT -- Microsoft
 ********************************************************************
 * Programm: MAIN
 * Datei: FB_MainUnwinderCtrl.st
 * Autor: Awalz
 * Erstellt: 7. April 2014
 ********************************************************************
 * Implementierung des Programms MAIN
 ********************************************************************)

 (*<$Description$> TODO: Bitte Kommentar hier einzufügen </$Description$>*)
FUNCTION_BLOCK FB_MainUnwinderCtrl
	unwinderOp.ctrl(BetrCtrl := BetrCtrl, machineaxis := machineaxis, unwinderaxis := unwinderOp.unwinderaxis, status := unwinderOp.status, buffertofull := buffertofull,
					 clamp := unwinderOp.clamp, lift := unwinderOp.lift, data := unwinderOp.data, clk := clk, webbuffer := webbuffer, IOs := IOs, panel := panel);
	unwinderOp.lift.enable :=  NOT unwinderDrv.lift.buttonDown AND NOT unwinderDrv.lift.buttonUp;
	unwinderDrv.ctrl(BetrCtrl := BetrCtrl,machineaxis := machineaxis, unwinderaxis := unwinderDrv.unwinderaxis,status := unwinderDrv.status, buffertofull := buffertofull,
						clamp := unwinderDrv.clamp,	lift := unwinderDrv.lift, data := unwinderDrv.data, clk := clk, webbuffer := webbuffer, IOs := IOs, panel := panel);
	unwinderDrv.lift.enable := NOT unwinderOp.lift.buttonDown AND NOT unwinderOp.lift.buttonUp;
	webbuffer();
	testpos := webbuffer.axis.ctrl.MC_ReadActualPosition_0.Position;
	feederCtrl(machineaxis := machineaxis, clk := clk);
	feederstatus(axisState := feederCtrl.MC_ReadStatus_0);
	clamp(clk := clk);
	splicetable(clk := clk);
	emcy_inputs();
//	data.undwinderDRV.recipeData.mode := CONST.UNITMODEs.ENABLE; (* später von der Visu oder dem Rezept freigeben*)
//	data.unwinderOP.recipeData.mode := CONST.UNITMODEs.ENABLE;
//	valveterminal.0 := unwinderOp.clamp.toDown_o;
//	valveterminal.7	:= splicetable.clampAfter.toDown_o;
//	valveterminal.1 := unwinderDrv.clamp.toDown_o;

	IF  panel.LDTRESET.LDT.button AND feederCtrl.MC_ReadStatus_0.Errorstop THEN (* prüfen*)
		feederCtrl.cmd := CONST.AXIS.RESET;
	END_IF

	CASE StateCtrl OF
		CTRL_FIRST_START:
		busy := TRUE;
		StateCtrl := CTRL_EMERGENCYSTOP_BEFORE;

	CTRL_MANUAL_BEFORE:
		IF BetrCtrl.value = CONST.MACHINEMODES.MANUAL THEN
			unwinderOp.ctrl.BetrCtrl(set := TRUE,value := CONST.MACHINEMODES.MANUAL);
			unwinderDrv.ctrl.BetrCtrl(set := TRUE,value := CONST.MACHINEMODES.MANUAL);
			IF NOT unwinderOp.ctrl.busy AND NOT unwinderDrv.ctrl.busy THEN
				BetrStatus(set := TRUE, value := BetrCtrl.value);
				busy := FALSE;
				err(reset := TRUE);
				state := ST_IDLE;
				StateCtrl := CTRL_MANUAL;
			END_IF
		ELSIF BetrCtrl.value = CONST.MACHINEMODES.EMERGENCYSTOP THEN
			StateCtrl := CTRL_EMERGENCYSTOP_BEFORE;
		ELSIF BetrCtrl.value = CONST.MACHINEMODES.SAFETYSTOP THEN
			StateCtrl := CTRL_SAFETYSTOP_BEFORE;
		ELSIF BetrCtrl.value = CONST.MACHINEMODES.AUTOMATIC THEN
			StateCtrl := CTRL_AUTO_BEFORE;
		END_IF

	CTRL_MANUAL:
		IF BetrCtrl.value <> CONST.MACHINEMODES.MANUAL THEN
			err(reset := TRUE);
			busy := TRUE;
			StateCtrl := CTRL_MANUAL_AFTER;
		ELSE
			ac_manualUnwinder; (*Aufruf der Action*)
		END_IF

	CTRL_MANUAL_AFTER:
		(*chkStatus.enable := FALSE;*)
		ac_setStateAfterUnwinder; (*Aufruf der Action*)

	CTRL_AUTO_BEFORE:
		IF BetrCtrl.value = CONST.MACHINEMODES.AUTOMATIC THEN
			BetrStatus(set := TRUE, value := CONST.MACHINEMODES.AUTOMATIC);
			(*clamp.init(clk := clk);
			chkStatus.enable := TRUE;*)
			err(reset := TRUE);
			busy := FALSE;
			state := ST_IDLE;
			StateCtrl := CTRL_AUTO;
		ELSIF BetrCtrl.value = CONST.MACHINEMODES.EMERGENCYSTOP THEN
			StateCtrl := CTRL_EMERGENCYSTOP_BEFORE;
		ELSIF BetrCtrl.value = CONST.MACHINEMODES.SAFETYSTOP THEN
			StateCtrl := CTRL_SAFETYSTOP_BEFORE;
		ELSIF BetrCtrl.value = CONST.MACHINEMODES.MANUAL THEN
			StateCtrl := CTRL_MANUAL_BEFORE;
		END_IF

	(* ******************************** *)
	(* *********** AUTO *************** *)
	(* ******************************** *)
	CTRL_AUTO:
		IF BetrCtrl.value <> CONST.MACHINEMODES.AUTOMATIC THEN
			err(reset := TRUE);
			busy := TRUE;
			StateCtrl := CTRL_AUTO_AFTER;
		ELSE
			ac_automUnwinder;
		END_IF

	CTRL_AUTO_AFTER:
		(*chkStatus.enable := FALSE;*)
		state := ST_IDLE;
		ac_setStateAfterUnwinder;

	CTRL_STOP_BEFORE:
		IF BetrCtrl.value = CONST.MACHINEMODES.EMERGENCYSTOP THEN
			StateCtrl := CTRL_EMERGENCYSTOP_BEFORE;
		ELSIF BetrCtrl.value = CONST.MACHINEMODES.SAFETYSTOP THEN
			StateCtrl := CTRL_SAFETYSTOP_BEFORE;
		ELSE
			state := ST_IDLE;
			StateCtrl := CTRL_STOP;
		END_IF

	CTRL_STOP:
		IF BetrCtrl.value = CONST.MACHINEMODES.EMERGENCYSTOP THEN
			StateCtrl := CTRL_EMERGENCYSTOP_BEFORE;
		ELSIF BetrCtrl.value = CONST.MACHINEMODES.SAFETYSTOP THEN
			StateCtrl := CTRL_SAFETYSTOP_BEFORE;
		ELSE
			CASE state OF
			ST_IDLE:
				state := ST_QUIT;

			ST_QUIT:
				state := ST_IDLE;
				StateCtrl := CTRL_STOP_AFTER;
			END_CASE
		END_IF

	CTRL_STOP_AFTER:
		IF BetrCtrl.value = CONST.MACHINEMODES.EMERGENCYSTOP THEN
			StateCtrl := CTRL_EMERGENCYSTOP_BEFORE;
		ELSIF BetrCtrl.value = CONST.MACHINEMODES.SAFETYSTOP THEN
			StateCtrl := CTRL_SAFETYSTOP_BEFORE;
		ELSIF BetrCtrl.value = CONST.MACHINEMODES.MANUAL THEN
			StateCtrl := CTRL_MANUAL_BEFORE;
		ELSIF BetrCtrl.value = CONST.MACHINEMODES.AUTOMATIC THEN
			StateCtrl := CTRL_AUTO_BEFORE;
		END_IF

	CTRL_RESET_START:
		BetrStatus(set := TRUE, value := CONST.MACHINEMODES.RESET);
		IF BetrCtrl.value = CONST.MACHINEMODES.EMERGENCYSTOP THEN
			StateCtrl := CTRL_EMERGENCYSTOP_BEFORE;
		ELSIF BetrCtrl.value = CONST.MACHINEMODES.SAFETYSTOP THEN
			StateCtrl := CTRL_SAFETYSTOP_BEFORE;
		ELSE
			feederCtrl.cmd := CONST.AXIS.POWER_OFF ;
			StateCtrl := CTRL_RESET;
		END_IF

	CTRL_RESET:
//		unwinderOp.unwinderaxis(machineaxis := machineaxis, dancer := unwinderOp.dancer, status := unwinderOp.status);
//		unwinderDrv.unwinderaxis(machineaxis := machineaxis, dancer := unwinderOp.dancer, status := unwinderOp.status);
		IF BetrCtrl.value = CONST.MACHINEMODES.EMERGENCYSTOP THEN
			StateCtrl := CTRL_EMERGENCYSTOP_BEFORE;
		ELSIF BetrCtrl.value = CONST.MACHINEMODES.SAFETYSTOP THEN
			StateCtrl := CTRL_SAFETYSTOP_BEFORE;
		ELSE
			StateCtrl := CTRL_RESET_AFTER;
		END_IF

	CTRL_RESET_AFTER:
		IF BetrCtrl.value = CONST.MACHINEMODES.RESET THEN
			busy := FALSE;
		ELSE
			busy := TRUE;
			(*clamp.init(clk := clk);
			err.reset();*)
			err(reset := TRUE);
			IF BetrCtrl.value = CONST.MACHINEMODES.EMERGENCYSTOP THEN
				StateCtrl := CTRL_EMERGENCYSTOP_BEFORE;
			ELSIF BetrCtrl.value = CONST.MACHINEMODES.SAFETYSTOP THEN
				StateCtrl := CTRL_SAFETYSTOP_BEFORE;
			ELSIF BetrCtrl.value = CONST.MACHINEMODES.SAFETYSTOP THEN
				StateCtrl := CTRL_SAFETYSTOP_BEFORE;
			ELSIF BetrCtrl.value = CONST.MACHINEMODES.MANUAL THEN
					feederCtrl.cmd := CONST.AXIS.POWER_ON ;
					StateCtrl := CTRL_MANUAL_BEFORE;
			ELSIF BetrCtrl.value = CONST.MACHINEMODES.AUTOMATIC THEN
					feederCtrl.cmd := CONST.AXIS.POWER_ON ;
					StateCtrl := CTRL_AUTO_BEFORE;
			END_IF
		END_IF

	CTRL_SAFETYSTOP_BEFORE:
		IF BetrCtrl.value = CONST.MACHINEMODES.EMERGENCYSTOP THEN
			StateCtrl := CTRL_EMERGENCYSTOP_BEFORE;
		ELSE
			BetrStatus.set := TRUE;
			BetrStatus.value := CONST.MACHINEMODES.SAFETYSTOP;
			state := ST_IDLE;
			StateCtrl := CTRL_SAFETYSTOP;
		END_IF

	CTRL_SAFETYSTOP:
		IF BetrCtrl.value = CONST.MACHINEMODES.EMERGENCYSTOP THEN
			StateCtrl := CTRL_EMERGENCYSTOP_BEFORE;
		ELSE
			CASE state OF
			ST_IDLE:
				IF NOT unwinderOp.ctrl.busy AND NOT unwinderDrv.ctrl.busy THEN
					state := ST_QUIT;
				END_IF
			ST_QUIT:
				state := ST_IDLE;
				BetrStatus(set := TRUE, value := CONST.MACHINEMODES.SAFETYSTOP);
				unwinderOp.ctrl.BetrCtrl(set := TRUE,value := CONST.MACHINEMODES.SAFETYSTOP);
				unwinderDrv.ctrl.BetrCtrl(set := TRUE,value := CONST.MACHINEMODES.SAFETYSTOP);
				feederCtrl.cmd := CONST.AXIS.POWER_OFF ;
				StateCtrl := CTRL_SAFETYSTOP_AFTER;
			END_CASE
		END_IF

	CTRL_SAFETYSTOP_AFTER:
		busy := FALSE;
		IF BetrCtrl.value = CONST.MACHINEMODES.EMERGENCYSTOP THEN
			busy := TRUE;
			StateCtrl := CTRL_EMERGENCYSTOP_BEFORE;
		ELSIF BetrCtrl.value = CONST.MACHINEMODES.MANUAL THEN
//			supplydelay(IN:= TRUE, PT := T#8s);
//				IF supplydelay.Q THEN
//					unwinderOp.unwinderaxis.cmd := CONST.AXIS.POWER_ON;
//					unwinderDrv.unwinderaxis.cmd := CONST.AXIS.POWER_ON;
//					busy := TRUE;
//					supplydelay(IN:= FALSE);
					feederCtrl.cmd := CONST.AXIS.POWER_ON ;
					StateCtrl := CTRL_MANUAL_BEFORE;
		ELSIF BetrCtrl.value = CONST.MACHINEMODES.AUTOMATIC THEN
//				supplydelay(IN:= TRUE, PT := T#8s);
//				IF supplydelay.Q THEN
//					unwinderOp.unwinderaxis.cmd := CONST.AXIS.POWER_ON;
//					unwinderDrv.unwinderaxis.cmd := CONST.AXIS.POWER_ON;
//					busy := TRUE;
//					supplydelay(IN:= FALSE);
					feederCtrl.cmd := CONST.AXIS.POWER_ON ;
					StateCtrl := CTRL_AUTO_BEFORE;
		END_IF

	CTRL_EMERGENCYSTOP_BEFORE:
		unwinderOp.ctrl.BetrCtrl(set := TRUE,value := CONST.MACHINEMODES.EMERGENCYSTOP);
		unwinderDrv.ctrl.BetrCtrl(set := TRUE,value := CONST.MACHINEMODES.EMERGENCYSTOP);
		(*axis.drvCtrl.resetRelease(ref := axis.ctrl.ref);*)
		IF NOT unwinderOp.ctrl.busy AND NOT unwinderDrv.ctrl.busy THEN

			IF unwinderOp.ctrl.BetrStatus.value = CONST.MACHINEMODES.EMERGENCYSTOP
				AND unwinderDrv.ctrl.BetrStatus.value = CONST.MACHINEMODES.EMERGENCYSTOP THEN
				BetrStatus(set := TRUE, value := CONST.MACHINEMODES.EMERGENCYSTOP);
				StateCtrl := CTRL_EMERGENCYSTOP;
			END_IF

		END_IF

	CTRL_EMERGENCYSTOP:
		IF BetrCtrl.value = CONST.MACHINEMODES.EMERGENCYSTOP THEN
			busy := FALSE;
		ELSE
			busy := TRUE;
			StateCtrl:= CTRL_RESET_START;
		END_IF

	END_CASE

END_FUNCTION_BLOCK
```

#### Package Logical/MainMachineCtrl/MAIN/MainUnwinding/Unwinder - Paket

#### ac_manualUnwinderCtrl.st
```iecst
(********************************************************************
 * COPYRIGHT -- Microsoft
 ********************************************************************
 * Programm: MAIN
 * Datei: ac_manualUnwinderCtrl.st
 * Autor: awalz
 * Erstellt: 24. Juni 2014
 ********************************************************************
 * Implementierung des Programms MAIN
 ********************************************************************)

(* Fügt eine neue Aktion zum IEC Programm oder Bibliothek *)
ACTION ac_manualUnwinderCtrl:
	CASE state OF
	ST_IDLE:
		IF BetrCtrl.value <> CONST.MACHINEMODES.MANUAL THEN
			state := ST_IDLE;
			err(reset := TRUE);
			busy := TRUE;
			status.ready := FALSE;
			StateCtrl := CTRL_MANUAL_AFTER;
		ELSE
			IF unwinderaxis.MC_ReadStatus_0.Error OR unwinderaxis.MC_ReadStatus_0.Errorstop  THEN
				unwinderaxis.cmd := CONST.AXIS.RESET;
				cmd := CONST.AXIS.RESET;
				state := ST_AXIS_STOP;
			ELSE
				IF data.recipeData.mode = CONST.UNITMODEs.ENABLE THEN
					IF unwinderaxis.MC_ReadStatus_0.Disabled THEN
						unwinderaxis(cmd := CONST.AXIS.POWER_ON, machineaxis := machineaxis, data := data);
						state := ST_AXIS_ON;
					END_IF
					IF unwinderaxis.MC_ReadStatus_0.StandStill THEN
						unwinderaxis(cmd := CONST.AXIS.START, machineaxis := machineaxis, data := data);
						state := ST_AXIS_RUN;
					END_IF
				ELSIF data.recipeData.mode =  CONST.UNITMODEs.DISABLE THEN
					IF unwinderaxis.MC_ReadStatus_0.Disabled THEN
						unwinderaxis(cmd := CONST.AXIS.POWER_ON, machineaxis := machineaxis, data := data);
						state := ST_AXIS_ON_DIS;
					ELSE
						unwinderaxis(cmd := CONST.AXIS.STOP, machineaxis := machineaxis, data := data);
						state := ST_AXIS_STOP;
					END_IF
				ELSIF  data.recipeData.mode = CONST.UNITMODEs.AXIS_OFF THEN
					unwinderaxis(cmd := CONST.AXIS.POWER_OFF, machineaxis := machineaxis, data := data);
					state := ST_AXIS_OFF;
				END_IF
			END_IF
		END_IF

	ST_AXIS_STOP:
			IF data.recipeData.mode <> CONST.UNITMODEs.DISABLE THEN
				state := ST_IDLE;
			END_IF

	ST_AXIS_ON_DIS:
			IF data.recipeData.mode = CONST.UNITMODEs.DISABLE THEN
				state := ST_IDLE;
			END_IF

	ST_AXIS_RUN:
			IF data.recipeData.mode <> CONST.UNITMODEs.ENABLE (*AND NOT unwinderaxis.MC_ReadStatus_0.StandStill *) THEN
				state := ST_IDLE;
			END_IF

	ST_AXIS_ON:
//			IF data.recipeData.mode = CONST.UNITMODEs.ENABLE THEN
//				state := ST_IDLE;
//			END_IF
			IF data.recipeData.mode = CONST.UNITMODEs.ENABLE THEN
				state := ST_IDLE;
			ELSIF data.recipeData.mode	<> CONST.UNITMODEs.ENABLE AND unwinderaxis.MC_ReadStatus_0.ContinuousMotion THEN
				state := ST_IDLE;
			END_IF
	ST_AXIS_OFF:
			IF data.recipeData.mode <> CONST.UNITMODEs.AXIS_OFF THEN
				state := ST_IDLE;
			END_IF

	END_CASE

END_ACTION
```

#### FB_UnwinderAxis.st - TODO: hier wird der Betriebmodus umgeschalten
```iecst
(********************************************************************
 * COPYRIGHT -- Microsoft
 ********************************************************************
 * Library: UserSpilke
 * Datei: FB_MainUnwiningCtrl.st
 * Autor: Awalz
 * Erstellt: 24. März 2014
 ********************************************************************
 * Implementierung der Library UserSpilke
 ********************************************************************)

(* TODO: hier wird der Betriebmodus umgeschalten *)
FUNCTION_BLOCK FB_UnwinderAxis
	IF firststart THEN
		pAxis ACCESS AxisREF;
		UnwinderSysPara.wndWidth		:= 550;	// [mm]
		UnwinderSysPara.minDiam			:= 76; //gMachRecipe.Winders.CoreDiam; // [mm]
		UnwinderSysPara.xDiam			:= 1000; //gMachRecipe.Winders.CoreDiam; // [mm]
		UnwinderSysPara.maxDiam			:= 1200; // [mm]
		UnwinderSysPara.minDiam			:= 76;	// [mm]
		UnwinderSysPara.minInertia		:= 1.0; // [kgm^2]
		UnwinderSysPara.xInertia		:= 1.0; // [kgm^2]
		UnwinderSysPara.gearRatio		:= 8; //GEAR_RATIO_UNWINDER; // [1]
		UnwinderSysPara.kvTorque		:= 0.01; // [Nms]
		UnwinderSysPara.posTorque		:= 0.1; // [Nm]
		UnwinderSysPara.negTorque		:= 0.1; // [Nm]
		UnwinderSysPara.matThickness	:= 50.00; // [um]
		UnwinderSysPara.wndWidth		:= 1000.00; // [mm]
		UnwinderSysPara.lineUnits		:= 1000000; // [units/m]
		UnwinderSysPara.wndUnits		:= pAxis.encoder_if.parameter.scaling.load.units; //gUnwinder.encoder_if.parameter.scaling.load.units; 	// [units]
		UnwinderSysPara.revMotor		:= pAxis.encoder_if.parameter.scaling.load.rev_motor; // gUnwinder.encoder_if.parameter.scaling.load.rev_motor; // [units]
		UnwinderSysPara.axisType		:= 1; // unwinder
		// set estimation parameters
		UnwinderEstPara.cycEstTrig 		:= 1000; // [units]
		UnwinderEstPara.cycEstWindow 	:= 1000; // [units]
		UnwinderEstPara.filterMode 		:= 2; // LQ filter
		UnwinderEstPara.filterWindow 	:= 3000; // 3 times cycEstTrig
		WNCCalcDiam_Unwinder.startDiam 		:= 500; // estimation of start diameter in [mm]
		WNCCalcDiam_Unwinder.setStartDiam 	:= TRUE; // set startDiam when FB is enabled
		WNCCalcDiam_Unwinder.pSysPara		:= ADR(UnwinderSysPara);
		WNCCalcDiam_Unwinder.pEstPara		:= ADR(UnwinderEstPara);
		//**************************************************************
		//**************	speed and torque feed forward ****************
		WNCCalcFFCtrl_Unwinder.uppTrqLimit		:= UDINT_TO_REAL (data.recipeData.maxDiamTension); (*.100;*)
		WNCCalcFFCtrl_Unwinder.lowTrqLimit		:= UDINT_TO_REAL (data.recipeData.minDiamTension);
		WNCCalcFFCtrl_Unwinder.pSysPara			:= ADR(UnwinderSysPara);
		//****************************************************************
		//**************	set parameters for dancer controller ****************
		UnwinderPidPara.Kp 						:= 0.1; // [1/s]
		UnwinderPidPara.Tn 						:= 1.0; // [s]
		UnwinderPidPara.Td 						:= 0.0; // [s]
		UnwinderPidPara.Tf 						:= 0.0; // [s]
		UnwinderPidPara.yi_max 					:= 500.0; // [mm/s]
		UnwinderPidPara.y_max 					:= 500.0; // [mm/s]
		UnwinderPidPara.y_min 					:= -500.0; // [mm/s]
		WNCProcessCtrl_Unwinder.gain 			:= 1.0; // [1]
		WNCProcessCtrl_Unwinder.setProcVar 		:= 12000.0; // [mm]
		WNCProcessCtrl_Unwinder.pSysPara		:= ADR(UnwinderSysPara);
		WNCProcessCtrl_Unwinder.pPidPara		:= ADR(UnwinderPidPara);
		//***********************************************************************
		//******** set parameters for linear interpolation of speed controller *************
		vecD[0]		:= UnwinderSysPara.minDiam;		// [mm]
		vecD[1]		:= 1200.0;		// [mm]
		vecD[2]		:= 0.0;
		vecKV[0]	:= 2.7;	// [As]
		vecKV[1]	:= 80.0;	// [As]
		vecKV[2]	:= 0.0;
		vecTN[0]	:= 0.00;	// [s]
		vecTN[1]	:= 0.15;	// [s]
		vecTN[2]	:= 0.0;
		WNCLipSctrlPara_Unwinder.pSysPara		:= ADR(UnwinderSysPara);
		WNCLipSctrlPara_Unwinder.numPoints		:= 2;
		WNCLipSctrlPara_Unwinder.pVecDiam		:= ADR(vecD);
		WNCLipSctrlPara_Unwinder.pVecSctrlKV	:= ADR(vecKV);
		WNCLipSctrlPara_Unwinder.pVecSctrlTN	:= ADR(vecTN);
		//**********************************************************************************
		//**************	set parameters for speed controller **************
		MC_BR_VelocityControl_Unwinder.Axis			:=  AxisREF;// ADR(gUnwinder);
		MC_BR_VelocityControl_Unwinder.Acceleration	:= 10000;
		MC_BR_VelocityControl_Unwinder.Deceleration	:= 10000;
		MC_BR_VelocityControl_Unwinder.TorqueMode	:= mcFF;
		//***********************************************************************
		firststart := FALSE;
	 END_IF
	//***********************************************************************
	masteraxisREF ACCESS machineaxis.AxisREF;
	MC_ReadActualPosition_0.Enable := NOT(MC_ReadActualPosition_0.Error);
	MC_ReadActualPosition_0.Axis := AxisREF;
	MC_ReadActualPosition_0();

	MC_BR_ReadDriveStatus_0.Axis			:= AxisREF;
	MC_BR_ReadDriveStatus_0.AdrDriveStatus	:= ADR(BasicControl.Status.DriveStatus); (*DriveStatus;*)
	MC_BR_ReadDriveStatus_0.Enable			:= NOT MC_BR_ReadDriveStatus_0.Error; (*MC_BR_ReadDriveStatus_0.Error;*)
	MC_BR_ReadDriveStatus_0();
	status.ready := NOT MC_BR_ReadDriveStatus_0.Error AND MC_BR_ReadDriveStatus_0.Valid AND NOT MC_BR_VelocityControl_Unwinder.Error;
	//**********	diameter estimation		****************
	WNCCalcDiam_Unwinder.enable			:= TRUE;
	WNCCalcDiam_Unwinder.actLinePos 	:=  REAL_TO_DINT (masteraxisREF.monitor.s); (* Strecke der Masterachse (Virtuelle Achse*)
	WNCCalcDiam_Unwinder.actDcrPos		:= 0; // gMachine.IO.AIn.DancerPos.Value.RawInt;
	WNCCalcDiam_Unwinder.actWndPos 		:= REAL_TO_DINT (MC_ReadActualPosition_0.Position);  (* Position der Abwicklerachse*)
	WNCCalcDiam_Unwinder.mode			:= TRUE;		// cyclic position based estimation mode
	WNCCalcDiam_Unwinder.setStartDiam	:= TRUE;(* BetrCtrl.enable; (*gMachine.Status.mAutoModeActive;*)
	WNCCalcDiam_Unwinder();
	//************   limit diameter ******************************
	LCRLimit_0.min_value				:= 76;
	LCRLimit_0.max_value				:= 1500;
	LCRLimit_0.in						:= WNCCalcDiam_Unwinder.actDiam;
	LCRLimit_0();
	//********************************************************

	//*********** torque feed forward ************************
	WNCCalcFFCtrl_Unwinder.enable			:= TRUE;
	WNCCalcFFCtrl_Unwinder.sync				:= TRUE;	// sync. winder set speed with line speed
	WNCCalcFFCtrl_Unwinder.setMatTension	:= 0.0;
	WNCCalcFFCtrl_Unwinder.setLineSpeed 	:= machineaxis.MC_ReadActualVelocity_0.Velocity; (*AxisIf.Status.ActMasterVelocity;*)
	WNCCalcFFCtrl_Unwinder.actDiam 			:= LCRLimit_0.out;
	WNCCalcFFCtrl_Unwinder.actInertia 		:= WNCCalcDiam_Unwinder.actInertia;
	WNCCalcFFCtrl_Unwinder();
	//********************************************************
	MC_BR_VelocityControl_Unwinder.CyclicVelocityCorrection	:= WNCProcessCtrl_Unwinder.actSpeedCorr;
	MC_BR_VelocityControl_Unwinder.CyclicTorque				:= WNCCalcFFCtrl_Unwinder.setMotorTrq;
	MC_BR_VelocityControl_Unwinder.CyclicVelocity			:= WNCCalcFFCtrl_Unwinder.setWndSpeed;
	MC_BR_VelocityControl_Unwinder.SctrlKv					:= WNCLipSctrlPara_Unwinder.actSctrlKV;
	MC_BR_VelocityControl_Unwinder.SctrlTn					:= WNCLipSctrlPara_Unwinder.actSctrlTN;
	MC_BR_VelocityControl_Unwinder();
	//*********** dancer controller **************************
	WNCProcessCtrl_Unwinder.enable			:= TRUE;
	WNCProcessCtrl_Unwinder.actProcVar		:= INT_TO_REAL (0);  (* Istposition des Tänzers*)
	WNCProcessCtrl_Unwinder.actDiam			:= LCRLimit_0.out;
	WNCProcessCtrl_Unwinder.setProcVar 		:= data.recipeData.dancersolPos;				(* soll Position des Tänzers*)
	WNCProcessCtrl_Unwinder();
	//********************************************************
	//************** linear interpolation of speed controller  *************************
	WNCLipSctrlPara_Unwinder.enable			:= TRUE;
	WNCLipSctrlPara_Unwinder.actDiam		:= LCRLimit_0.out;
	WNCLipSctrlPara_Unwinder();
	//***********************************************************************************

	IF cmd = CONST.AXIS.POWER_ON THEN
		MC_Power_0.Enable := TRUE;
		IF MC_Power_0.Status THEN
			cmdtmp := cmd;
			cmd := CONST.AXIS.NOACTION;
		END_IF
	ELSIF cmd = CONST.AXIS.POWER_OFF THEN
		MC_Power_0.Enable := FALSE;
		MC_BR_VelocityControl_Unwinder.Enable := FALSE;
		IF NOT MC_Power_0.Status THEN
			cmdtmp := cmd;
			cmd:= CONST.AXIS.NOACTION;
		END_IF
	ELSIF cmd = CONST.AXIS.RESET THEN
		MC_Reset_0.Execute := TRUE;
		IF MC_Reset_0.Done THEN
			MC_Reset_0.Execute := FALSE;
			cmdtmp := cmd;
			cmd:= CONST.AXIS.NOACTION;
		END_IF

	END_IF

	IF cmd = CONST.AXIS.START THEN
		(*MC_Power_0.Enable := TRUE;*)
		(*IF MC_Power_0.Status AND NOT MC_Power_0.Error THEN *)
			MC_BR_VelocityControl_Unwinder.Enable := TRUE;
//			MC_BR_VelocityControl_Unwinder.CyclicVelocity			:= - WNCCalcFFCtrl_Unwinder.setWndSpeed;
//			MC_BR_VelocityControl_Unwinder.CyclicVelocityCorrection	:= - WNCProcessCtrl_Unwinder.actSpeedCorr;
//			MC_BR_VelocityControl_Unwinder.CyclicTorque				:= WNCCalcFFCtrl_Unwinder.setMotorTrq;
//
//			MC_Stop_0.Execute := FALSE;
//		ELSIF NOT  MC_Power_0.Status THEN
//			MC_Power_0.Enable := TRUE;
//		END_IF
	(*	cmd := CONST.AXIS.NOACTION;*)
	ELSIF cmd = CONST.AXIS.STOP THEN
		(*MC_Power_0.Enable :=FALSE;*)
		(*MC_Power_0.Enable := FALSE;*)
		MC_BR_VelocityControl_Unwinder.Enable := FALSE;
		MC_BR_VelocityControl_Unwinder.CyclicVelocityCorrection := 0;
		MC_BR_VelocityControl_Unwinder.CyclicTorque				:= 0;
		MC_BR_VelocityControl_Unwinder.CyclicVelocity			:= 0;
	(*	MC_Stop_0.Execute := TRUE;*)

	(*	cmd := CONST.AXIS.NOACTION;*)
	END_IF

//	CASE AxisStep OF
//	(******************* WAIT *************************)
//	(*	STATE_WAIT:  (* STATE: Wait *)
//	STATE_WAIT:  (* STATE: Waiting FOR commands *)
//		IF cmd <> CONST.AXIS.NOACTION THEN
//					busy := TRUE;
//					cmdtmp:= cmd;
//					IF cmd = CONST.AXIS.RESET THEN
//						AxisStep := STATE_ERROR_RESET;
//					ELSIF cmd = CONST.AXIS.STOP THEN
//						MC_Stop_0( Execute := TRUE, Deceleration := verzoegerung);
//						AxisStep := STATE_STOP;
//					ELSIF cmd = CONST.AXIS.START THEN
//						AxisStep := STATE_MOVE_VELOCITY;
//					ELSIF   cmd = CONST.AXIS.POWER_OFF THEN
//						AxisStep := STATE_POWER_OFF;
//					ELSIF   cmd = CONST.AXIS.POWER_ON THEN
//						AxisStep := STATE_POWER_ON;
//					END_IF
//		ELSE
//			busy := FALSE;
//		END_IF
//
//	STATE_POWER_ON:
//		IF cmd = CONST.AXIS.POWER_ON AND NOT MC_Power_0.Error AND NOT
//			 MC_Power_0.Status AND NOT MC_ReadStatus_0.Error  AND NOT MC_ReadStatus_0.Errorstop  THEN
//			MC_Power_0.Enable := TRUE;
//			cmd := cmdtmp;
////		ELSIF MC_Power_0.Error THEN
////			MC_Power_0.Enable := FALSE;
////			cmd := cmdtmp;
////			AxisStep := STATE_ERROR_RESET;
//				(*	merker := TRUE;  *)
//		ELSIF MC_Power_0.Status AND NOT MC_Power_0.Error THEN
//				cmdtmp := cmd;
//				AxisStep := STATE_QUIT;
////		ELSIF MC_ReadStatus_0.Error  OR MC_ReadStatus_0.Errorstop OR MC_Power_0.Error THEN
////			cmd := cmdtmp;
////			AxisStep := STATE_ERROR_RESET;
//	END_IF
////
//	STATE_POWER_OFF:
//		IF 	cmd = CONST.AXIS.POWER_OFF THEN
//			MC_Power_0.Enable := FALSE;
//			cmd := cmdtmp;
//			AxisStep := STATE_QUIT;
//		END_IF
////
//	STATE_ERROR_RESET:
//			MC_Power_0.Enable := FALSE;
//			MC_BR_VelocityControl_Unwinder.Enable := FALSE;
//			IF MC_Power_0.Error OR MC_BR_VelocityControl_Unwinder.Error
//				OR MC_ReadStatus_0.Error OR MC_ReadStatus_0.Errorstop  THEN
//				MC_Reset_0.Execute := TRUE;
//			ELSIF MC_Reset_0.Done THEN
//				MC_Reset_0.Execute := FALSE;
//				cmd := cmdtmp;
//				AxisStep := STATE_QUIT;
//			ELSIF (MC_ReadStatus_0.Disabled OR MC_ReadStatus_0.StandStill OR MC_ReadStatus_0.ContinuousMotion ) AND (NOT  MC_Power_0.Error
//				AND NOT  MC_BR_VelocityControl_Unwinder.Error AND NOT MC_ReadStatus_0.Error AND NOT  MC_ReadStatus_0.Errorstop) THEN (* axis is ok*)
//				MC_Reset_0.Execute := FALSE;
//				cmd := cmdtmp;
//				AxisStep := STATE_QUIT;
//			END_IF
////
//	STATE_QUIT:
//		IF cmd = cmdtmp THEN
//			cmd := CONST.AXIS.NOACTION;
//			AxisStep := STATE_WAIT;
//		ELSIF cmd <> CONST.AXIS.NOACTION THEN
//			AxisStep := STATE_WAIT;
//		END_IF
////
//	STATE_MOVE_VELOCITY:
//	//************************* speed controller  ************************************
//		IF cmd = CONST.AXIS.START AND NOT  MC_BR_VelocityControl_Unwinder.Error THEN
//			MC_BR_VelocityControl_Unwinder.Enable := TRUE;
//			MC_BR_VelocityControl_Unwinder.CyclicVelocityCorrection	:= WNCProcessCtrl_Unwinder.actSpeedCorr;
//			MC_BR_VelocityControl_Unwinder.CyclicTorque				:= WNCCalcFFCtrl_Unwinder.setMotorTrq;
//			MC_BR_VelocityControl_Unwinder.CyclicVelocity			:= WNCCalcFFCtrl_Unwinder.setWndSpeed;
//			MC_Stop_0.Execute := FALSE;
//			cmd := cmdtmp;
////		ELSIF MC_BR_VelocityControl_Unwinder.Error THEN
////			AxisStep := STATE_ERROR_RESET;
//		ELSIF cmd <> CONST.AXIS.START THEN
//			AxisStep := STATE_QUIT;
//		END_IF
////
//	STATE_STOP:
//		IF cmd = CONST.AXIS.STOP OR  MC_BR_VelocityControl_Unwinder.Error THEN
//			MC_BR_VelocityControl_Unwinder.Enable := FALSE;
//			MC_BR_VelocityControl_Unwinder.CyclicVelocityCorrection := 0;
//			MC_BR_VelocityControl_Unwinder.CyclicTorque				:= 0;
//			MC_BR_VelocityControl_Unwinder.CyclicVelocity			:= 0;
//			MC_Stop_0.Execute := TRUE;
//			cmdtmp := cmd;
//			IF MC_Stop_0.Done THEN
//				MC_Stop_0.Execute := FALSE;
//				AxisStep := STATE_QUIT;
//			END_IF
//		ELSIF MC_BR_VelocityControl_Unwinder.Error THEN
//			AxisStep := STATE_ERROR_RESET;
//		END_IF
//
//	END_CASE

	(************************ MC_READSTATUS *************************)
	MC_ReadStatus_0.Enable :=  NOT MC_ReadStatus_0.Error;
	MC_ReadStatus_0.Axis := AxisREF;
	MC_ReadStatus_0();
	(************************** MC_POWER ****************************)
	MC_Power_0.Axis := AxisREF;  (* pointer to axis *)
	MC_Power_0();

	(************************** MC_STOP *****************************)
	MC_Stop_0.Axis := AxisREF;
	MC_Stop_0();
	(***************************MC_HALT******************************)
	(*MC_Halt_0.Axis := AxisREF;
	MC_Halt_0();
	(************************** MC_RESET ****************************)
	MC_Reset_0.Axis := AxisREF;
	MC_Reset_0();
END_FUNCTION_BLOCK
```

#### ac_automUnwinderCtrl.st
```iecst
(********************************************************************
 * COPYRIGHT -- Microsoft
 ********************************************************************
 * Programm: MAIN
 * Datei: ac_automUnwinderCtrl.st
 * Autor: awalz
 * Erstellt: 24. Juli 2014
 ********************************************************************
 * Implementierung des Programms MAIN
 ********************************************************************)

(* Fügt eine neue Aktion zum IEC Programm oder Bibliothek *)
ACTION ac_automUnwinderCtrl:

	CASE state OF
		ST_IDLE:
			IF BetrCtrl.value <> CONST.MACHINEMODES.AUTOMATIC THEN
				state := ST_IDLE;
				err(reset := TRUE);
				busy := TRUE;
				status.ready := FALSE;
				StateCtrl := CTRL_AUTO_AFTER;
			ELSE
				IF unwinderaxis.MC_ReadStatus_0.Error OR unwinderaxis.MC_ReadStatus_0.Errorstop  THEN
					unwinderaxis.cmd := CONST.AXIS.RESET;
					cmd := CONST.AXIS.RESET;
					state := ST_AXIS_STOP;
				ELSE
					IF data.recipeData.mode = CONST.UNITMODEs.ENABLE THEN
						IF unwinderaxis.MC_ReadStatus_0.Disabled THEN
							unwinderaxis(cmd := CONST.AXIS.POWER_ON, machineaxis := machineaxis, data := data);
							state := ST_AXIS_ON;
						END_IF
						IF unwinderaxis.MC_ReadStatus_0.StandStill THEN
							unwinderaxis(cmd := CONST.AXIS.START, machineaxis := machineaxis, data := data);
							state := ST_AXIS_RUN;
						END_IF
					ELSIF data.recipeData.mode =  CONST.UNITMODEs.DISABLE THEN
						IF unwinderaxis.MC_ReadStatus_0.Disabled THEN
							unwinderaxis(cmd := CONST.AXIS.POWER_ON, machineaxis := machineaxis, data := data);
							state := ST_AXIS_ON_DIS;
						ELSE
							unwinderaxis(cmd := CONST.AXIS.STOP, machineaxis := machineaxis, data := data);
							state := ST_AXIS_STOP;
						END_IF
					ELSIF  data.recipeData.mode = CONST.UNITMODEs.AXIS_OFF THEN
						unwinderaxis(cmd := CONST.AXIS.POWER_OFF, machineaxis := machineaxis, data := data);
						state := ST_AXIS_OFF;
					END_IF
				END_IF
			END_IF

		ST_AXIS_STOP:
				IF data.recipeData.mode <> CONST.UNITMODEs.DISABLE THEN
					state := ST_IDLE;
				END_IF

		ST_AXIS_ON_DIS:
				IF data.recipeData.mode = CONST.UNITMODEs.DISABLE THEN
					state := ST_IDLE;
				END_IF

		ST_AXIS_RUN:
				IF data.recipeData.mode <> CONST.UNITMODEs.ENABLE (*AND NOT unwinderaxis.MC_ReadStatus_0.StandStill *) THEN
					state := ST_IDLE;
				END_IF

		ST_AXIS_ON:
				IF data.recipeData.mode = CONST.UNITMODEs.ENABLE THEN
					state := ST_IDLE;
				END_IF

		ST_AXIS_OFF:
				IF data.recipeData.mode <> CONST.UNITMODEs.AXIS_OFF THEN
					state := ST_IDLE;
				END_IF

	END_CASE
END_ACTION
```

#### FB_UnwinderCtrl.st
```iecst
(********************************************************************
 * COPYRIGHT -- Microsoft
 ********************************************************************
 * Programm: MAIN
 * Datei: FB_UnwinderCtrl.st
 * Autor: awalz
 * Erstellt: 24. Juni 2014
 ********************************************************************
 * Implementierung des Programms MAIN
 ********************************************************************)

(* TODO: Bitte Kommentar hier einfügen *)
FUNCTION_BLOCK FB_UnwinderCtrl
	(* nicht vergessen die Sollposition des Bahnpuffers vorgeben*)
	webbuffer();(* die Lage des Bahnspeichers für die Kraftumschaltung*)
	IOs(panel := panel);(* Abfrage ob die die Maschine im Inlinemode ist*)
	unwinderaxis(machineaxis := machineaxis, data := data,startdiameter := 560);
//	unwinderaxis.WNCCalcDiam_0.actDcrPos := webbuffer.axis.ctrl.MC_ReadActualPosition_0.Position/1000;
	status.ready := (unwinderaxis.MC_ReadStatus_0.ContinuousMotion OR unwinderaxis.MC_ReadStatus_0.StandStill) AND NOT unwinderaxis.MC_ReadStatus_0.Disabled;
	status(axisState := unwinderaxis.MC_ReadStatus_0);
	(*dancer();*)
	clamp( clk := clk);
	testpos := webbuffer.axis.ctrl.MC_ReadActualPosition_0.Position;

	unwinderaxis.bufferUpDownKeys := webbuffer.keys.up.LDT.button OR webbuffer.keys.down.LDT.button; // Abfrage der hoch und runter Tasten des Bahnspeichers //OKrebs 16.09.14

	buffertofullRtrig(CLK := IOs.inline (*OR buffertofull*));
	IF IOs.inline THEN
		IF buffertofullRtrig.Q AND webbuffer.axis.ctrl.MC_ReadActualPosition_0.Position < 5800 THEN (* Position gilt noch zu definieren*)
			unwinderaxis.mode := TRUE;
		ELSIF buffertofull AND webbuffer.axis.ctrl.MC_ReadActualPosition_0.Position < 5800 THEN
			unwinderaxis.mode := TRUE;
		ELSIF  webbuffer.axis.ctrl.MC_ReadActualPosition_0.Position > 5800 THEN
			unwinderaxis.mode := FALSE;
		END_IF
	ELSE
		unwinderaxis.mode := FALSE;
	END_IF
	IF data.recipeData.mode = CONST.UNITMODEs.ENABLE THEN
		IF data.recipeData.warnDiam > unwinderaxis.LCRLimit_0.out  THEN
			diameterWarning := TRUE;
		ELSE
			diameterWarning := FALSE;
		END_IF
		IF data.recipeData.stopDiam > unwinderaxis.LCRLimit_0.out THEN
			diameterStop := TRUE;
		ELSE
			diameterStop := FALSE;
		END_IF
//		diameterStop := SEL((data.recipeData.stopDiam > unwinderaxis.WNCCalcDiam_0.actDiam AND unwinderaxis.WNCCalcDiam_0.actDiam > 0 ), FALSE, TRUE);
//		diameterWarning := SEL ((data.recipeData.warnDiam > unwinderaxis.WNCCalcDiam_0.actDiam AND unwinderaxis.WNCCalcDiam_0.actDiam > 0), FALSE, TRUE);
	ELSE
		diameterStop := FALSE;
		diameterWarning := FALSE;
	END_IF
(*	data.recipeData.mode := CONST.UNITMODEs.ENABLE; *)(* später von der Visu oder dem Rezept freigeben*)
	lift();
CASE StateCtrl OF
	CTRL_FIRST_START:
		busy := TRUE;
		StateCtrl := CTRL_EMERGENCYSTOP_BEFORE;

	CTRL_MANUAL_BEFORE:
		IF BetrCtrl.value = CONST.MACHINEMODES.MANUAL THEN
			BetrStatus(set := TRUE,value := CONST.MACHINEMODES.MANUAL);
			busy := FALSE;
			(*clamp.init(clk := clk);*)
			(*chkStatus.enable := TRUE;*)
			err(reset := TRUE);
			timer(IN:= FALSE);
			state := ST_IDLE;
			firstStart := TRUE;
			StateCtrl := CTRL_MANUAL;
		ELSIF BetrCtrl.value = CONST.MACHINEMODES.EMERGENCYSTOP THEN
			StateCtrl := CTRL_EMERGENCYSTOP_BEFORE;
		ELSIF BetrCtrl.value = CONST.MACHINEMODES.SAFETYSTOP THEN
			StateCtrl := CTRL_SAFETYSTOP_BEFORE;
		ELSIF BetrCtrl.value = CONST.MACHINEMODES.AUTOMATIC THEN
			StateCtrl := CTRL_AUTO_BEFORE;
		END_IF

	CTRL_MANUAL:
		IF BetrCtrl.value <> CONST.MACHINEMODES.MANUAL THEN
			err(reset := TRUE);
			busy := TRUE;
			StateCtrl := CTRL_MANUAL_AFTER;
		ELSE
			ac_manualUnwinderCtrl; (*Aufruf der Action*)
		END_IF

	CTRL_MANUAL_AFTER:
		(*chkStatus.enable := FALSE;*)
		ac_setStateAfterUnwinder; (*Aufruf der Action*)

	CTRL_AUTO_BEFORE:
		IF BetrCtrl.value = CONST.MACHINEMODES.AUTOMATIC THEN
			BetrStatus(set := TRUE, value := CONST.MACHINEMODES.AUTOMATIC);
			err(reset := TRUE);
			busy := FALSE;
			state := ST_IDLE;
			StateCtrl := CTRL_AUTO;
		ELSIF BetrCtrl.value = CONST.MACHINEMODES.EMERGENCYSTOP THEN
			StateCtrl := CTRL_EMERGENCYSTOP_BEFORE;
		ELSIF BetrCtrl.value = CONST.MACHINEMODES.SAFETYSTOP THEN
			StateCtrl := CTRL_SAFETYSTOP_BEFORE;
		ELSIF BetrCtrl.value = CONST.MACHINEMODES.MANUAL THEN
			StateCtrl := CTRL_MANUAL_BEFORE;
		END_IF

	(* ******************************** *)
	(* *********** AUTO *************** *)
	(* ******************************** *)
	CTRL_AUTO:
		IF BetrCtrl.value <> CONST.MACHINEMODES.AUTOMATIC THEN
			err(reset := TRUE);
			busy := TRUE;
			StateCtrl := CTRL_AUTO_AFTER;
		ELSE
			ac_automUnwinderCtrl;
		END_IF

	CTRL_AUTO_AFTER:
		(*chkStatus.enable := FALSE;*)
		state := ST_IDLE;
		ac_setStateAfterUnwinder;

	CTRL_STOP_BEFORE:
		IF BetrCtrl.value = CONST.MACHINEMODES.EMERGENCYSTOP THEN
			StateCtrl := CTRL_EMERGENCYSTOP_BEFORE;
		ELSIF BetrCtrl.value = CONST.MACHINEMODES.SAFETYSTOP THEN
			StateCtrl := CTRL_SAFETYSTOP_BEFORE;
		ELSE
			state := ST_IDLE;
			StateCtrl := CTRL_STOP;
		END_IF

	CTRL_STOP:
		IF BetrCtrl.value = CONST.MACHINEMODES.EMERGENCYSTOP THEN
			StateCtrl := CTRL_EMERGENCYSTOP_BEFORE;
		ELSIF BetrCtrl.value = CONST.MACHINEMODES.SAFETYSTOP THEN
			StateCtrl := CTRL_SAFETYSTOP_BEFORE;
		ELSE
			CASE state OF
			ST_IDLE:
				state := ST_QUIT;

			ST_QUIT:
				state := ST_IDLE;
				StateCtrl := CTRL_STOP_AFTER;
			END_CASE
		END_IF

	CTRL_STOP_AFTER:
		IF BetrCtrl.value = CONST.MACHINEMODES.EMERGENCYSTOP THEN
			StateCtrl := CTRL_EMERGENCYSTOP_BEFORE;
		ELSIF BetrCtrl.value = CONST.MACHINEMODES.SAFETYSTOP THEN
			StateCtrl := CTRL_SAFETYSTOP_BEFORE;
		ELSIF BetrCtrl.value = CONST.MACHINEMODES.MANUAL THEN
			StateCtrl := CTRL_MANUAL_BEFORE;
		ELSIF BetrCtrl.value = CONST.MACHINEMODES.AUTOMATIC THEN
			StateCtrl := CTRL_AUTO_BEFORE;
		END_IF

	CTRL_RESET_START:
		BetrStatus.set := TRUE;
		BetrStatus.value := CONST.MACHINEMODES.RESET;
		IF BetrCtrl.value = CONST.MACHINEMODES.EMERGENCYSTOP THEN
			StateCtrl := CTRL_EMERGENCYSTOP_BEFORE;
		ELSIF BetrCtrl.value = CONST.MACHINEMODES.SAFETYSTOP THEN
			StateCtrl := CTRL_SAFETYSTOP_BEFORE;
		ELSE
			IF unwinderaxis.busy  OR unwinderaxis.cmd <> CONST.AXIS.NOACTION THEN
				unwinderaxis(cmd := CONST.AXIS.NOACTION, data := data, machineaxis := machineaxis, (*dancer := dancer,*) (*status := status*));
			ELSE
				unwinderaxis(cmd := CONST.AXIS.RESET, data := data, machineaxis := machineaxis, (*dancer := dancer,*)(* status := status*));
				StateCtrl := CTRL_RESET;
			END_IF
		END_IF

	CTRL_RESET:
		unwinderaxis(machineaxis := machineaxis, data := data, (*dancer := dancer,*)(* status := status*));
		IF BetrCtrl.value = CONST.MACHINEMODES.EMERGENCYSTOP THEN
			StateCtrl := CTRL_EMERGENCYSTOP_BEFORE;
		ELSIF BetrCtrl.value = CONST.MACHINEMODES.SAFETYSTOP THEN
			StateCtrl := CTRL_SAFETYSTOP_BEFORE;
		ELSE
			(*IF NOT unwinderaxis.busy THEN*)
				unwinderaxis.cmd := CONST.AXIS.POWER_OFF;
				StateCtrl := CTRL_RESET_AFTER;
			(*END_IF*)
		END_IF

	CTRL_RESET_AFTER:
		IF BetrCtrl.value = CONST.MACHINEMODES.RESET THEN
			busy := FALSE;
		ELSE
			busy := TRUE;
			(*clamp.init(clk := clk);
			err.reset();*)
			err(reset := TRUE);
			IF BetrCtrl.value = CONST.MACHINEMODES.EMERGENCYSTOP THEN
				StateCtrl := CTRL_EMERGENCYSTOP_BEFORE;
//			ELSIF BetrCtrl.value = CONST.MACHINEMODES.SAFETYSTOP THEN
//				StateCtrl := CTRL_SAFETYSTOP_BEFORE;
			ELSIF BetrCtrl.value = CONST.MACHINEMODES.SAFETYSTOP THEN
				StateCtrl := CTRL_SAFETYSTOP_BEFORE;
			ELSIF BetrCtrl.value = CONST.MACHINEMODES.MANUAL THEN
			supplydelay(IN:= TRUE, PT := T#8s);
				IF supplydelay.Q THEN
					unwinderaxis.cmd := CONST.AXIS.POWER_ON;
					busy := TRUE;
					supplydelay(IN:= FALSE);
					StateCtrl := CTRL_MANUAL_BEFORE;
				END_IF
			ELSIF BetrCtrl.value = CONST.MACHINEMODES.AUTOMATIC THEN
				supplydelay(IN:= TRUE, PT := T#8s);
				IF supplydelay.Q THEN
					unwinderaxis.cmd := CONST.AXIS.POWER_ON;
					busy := TRUE;
					supplydelay(IN:= FALSE);
					StateCtrl := CTRL_AUTO_BEFORE;
				END_IF
			END_IF
		END_IF

	CTRL_SAFETYSTOP_BEFORE:
		IF BetrCtrl.value = CONST.MACHINEMODES.EMERGENCYSTOP THEN
			StateCtrl := CTRL_EMERGENCYSTOP_BEFORE;
		ELSE
			BetrStatus.set := TRUE;
			BetrStatus.value := CONST.MACHINEMODES.SAFETYSTOP;
			unwinderaxis.cmd := CONST.AXIS.POWER_OFF;(* neue weil die Achse nicht ausgeschaltet wird*)
			state := ST_IDLE;
			StateCtrl := CTRL_SAFETYSTOP;
		END_IF

	CTRL_SAFETYSTOP:
		IF BetrCtrl.value = CONST.MACHINEMODES.EMERGENCYSTOP THEN
			StateCtrl := CTRL_EMERGENCYSTOP_BEFORE;
		ELSE
			CASE state OF
			ST_IDLE:
				unwinderaxis.cmd := CONST.AXIS.RESET;
				state := ST_QUIT;
			ST_QUIT:
				state := ST_QUIT;
				StateCtrl := CTRL_SAFETYSTOP_AFTER;
			END_CASE
		END_IF

	CTRL_SAFETYSTOP_AFTER:
		busy := FALSE;
		IF BetrCtrl.value = CONST.MACHINEMODES.EMERGENCYSTOP THEN
			busy := TRUE;
			StateCtrl := CTRL_EMERGENCYSTOP_BEFORE;
		ELSIF BetrCtrl.value = CONST.MACHINEMODES.MANUAL THEN
			supplydelay(IN:= TRUE, PT := T#8s);
				IF supplydelay.Q THEN
					unwinderaxis.cmd := CONST.AXIS.POWER_ON;
					busy := TRUE;
					supplydelay(IN:= FALSE);
					StateCtrl := CTRL_MANUAL_BEFORE;
				END_IF
		ELSIF BetrCtrl.value = CONST.MACHINEMODES.AUTOMATIC THEN
				supplydelay(IN:= TRUE, PT := T#8s);
				IF supplydelay.Q THEN
					unwinderaxis.cmd := CONST.AXIS.POWER_ON;
					busy := TRUE;
					supplydelay(IN:= FALSE);
					StateCtrl := CTRL_AUTO_BEFORE;
				END_IF
		END_IF

	CTRL_EMERGENCYSTOP_BEFORE:
		(*axis.drvCtrl.resetRelease(ref := axis.ctrl.ref);*)
		BetrStatus(set := TRUE,value := CONST.MACHINEMODES.EMERGENCYSTOP);
		(*mode.status.set(value := CONST.MACHINEMODES.EMERGENCYSTOP);*)
		busy := FALSE;
		StateCtrl := CTRL_EMERGENCYSTOP;

	CTRL_EMERGENCYSTOP:
		unwinderaxis.cmd := CONST.AXIS.POWER_OFF;
		IF BetrCtrl.value = CONST.MACHINEMODES.EMERGENCYSTOP THEN
			;
		ELSE
			busy := TRUE;
			timer(IN := TRUE, PT := T#2s);
			StateCtrl := CTRL_EMERGENCYSTOP_AFTER;
		END_IF

	CTRL_EMERGENCYSTOP_AFTER:
		timer();
		IF BetrCtrl.value = CONST.MACHINEMODES.EMERGENCYSTOP THEN
			timer(IN := FALSE);
			BetrStatus(set := TRUE,value := CONST.MACHINEMODES.EMERGENCYSTOP);
			busy := FALSE;
			StateCtrl := CTRL_EMERGENCYSTOP;
		ELSIF timer.Q THEN
			timer(IN := FALSE);
			StateCtrl := CTRL_RESET_START;
		END_IF

		ELSE
			;
	END_CASE

END_FUNCTION_BLOCK
```

#### FB_Dancer.st
```iecst
(********************************************************************
 * COPYRIGHT -- Microsoft
 ********************************************************************
 * Library: UserSpilke
 * Datei: FB_Dancer.st
 * Autor: Awalz
 * Erstellt: 25. März 2014
 ********************************************************************
 * Implementierung der Library UserSpilke
 ********************************************************************)

(* TODO: Bitte Kommentar hier einzufügen *)
FUNCTION_BLOCK FB_Dancer
//((DINT_TO_REAL (DMS_In )) - offset) * SCALE_DINT_TO_400N) das ist die tasächliche Kraft was auf die Messwalze wirkt.Die Kraft wurde mit Hilfe einer ZUgwaage validiert*)
// da auf jede Seite der Bahn nur die Hälfte der Kraft wirkt muss um richtigkeitshalber die Auflösung halbiert werden
	pos_out := INT_TO_REAL (Pos) *SCALE_INT_TO_200MM;
	tension_output := REAL_TO_INT (setTension /(SCALE_100N_TO_INT));
	tension_scaled := (((DINT_TO_REAL (DMS_In )) - offset) * SCALE_DINT_TO_400N) /2;

	FlengeDMS := CFG_FLENGE_DMS_AIN;
END_FUNCTION_BLOCK
```

#### Package Logical/MainMachineCtrl/MAIN/Webbuffer - Paket

#### ac_manualbufferCtrl.st
```iecst
(********************************************************************
 * COPYRIGHT -- Microsoft
 ********************************************************************
 * Programm: MAIN
 * Datei: ac_bufferCtrl.st
 * Autor: awalz
 * Erstellt: 10. Juli 2014
 ********************************************************************
 * Implementierung des Programms MAIN
 ********************************************************************)

(* Fügt eine neue Aktion zum IEC Programm oder Bibliothek *)
ACTION ac_manualbufferCtrl:
//	axis.bufferaxis(machineaxis := machineaxis, data := data); (*auskomentiert am 21.08.14*)
	config( axis := axis, status := status);
	IF keys.home.LDT.button THEN
		cmdCtrl.value := CONST.CUTTINGUNIT.CMDs.CALIBR;
	ELSE
		cmdCtrl.value := CONST.CUTTINGUNIT.CMDs.NO_CMD;
//	ELSIF keys.home.LDT.ftrig THEN
//		cmdCtrl.value := CONST.CUTTINGUNIT.CMDs.NO_CMD;
	END_IF

	CASE state OF
	ST_IDLE:
		IF BetrCtrl.value <> CONST.MACHINEMODES.MANUAL THEN
//			state := ST_IDLE;
//			err(reset := TRUE);
			busy := TRUE;
			StateCtrl := CTRL_MANUAL_AFTER;

		ELSE
			IF 	firstStart AND  NOT axis.ctrl.BasicControl.AxisState.Homed  AND cmdCtrl.value = CONST.CUTTINGUNIT.CMDs.CALIBR AND mechbrakeON_OFF THEN
				firstStart := FALSE;
				unwinderOFF := TRUE;
				state := ST_FUNCTION_START;
//
			ELSIF (cmdCtrl.value =  CONST.CUTTINGUNIT.CMDs.MOVEBW OR cmdCtrl.value =  CONST.CUTTINGUNIT.CMDs.MOVEFW)
				AND axis.ctrl.BasicControl.AxisState.Homed AND mechbrakeON_OFF THEN
					cmdStatus(set := TRUE, value := cmdCtrl.value);
					busy := TRUE;
//					unwinderOFF := TRUE;  //Auskommentiert weil: Beim hoch und runter bewegen soll der Abwickler an bleiben, OKrebs 16.09.14
					state := ST_MOVE_START;
			ELSE
			 	IF (*axis.ctrl.BasicControl.AxisState.Homed AND *) machineaxis.MC_ReadStatus_0.ContinuousMotion AND mechbrakeON_OFF
				AND cmdCtrl.value = CONST.CUTTINGUNIT.CMDs.NO_CMD THEN
					axis.bufferaxis.cmd := CONST.AXIS.START;
				ELSIF  (*machineaxis.MC_ReadStatus_0.StandStill OR*) cmdCtrl.value =  CONST.CUTTINGUNIT.CMDs.ABORT THEN
					axis.bufferaxis.cmd := CONST.AXIS.STOP;
				END_IF
//		END_IF
			END_IF
		END_IF

	ST_MOVE_START:
		IF cmdCtrl.value = CONST.CUTTINGUNIT.CMDs.NO_CMD THEN
			cmdStatus(set := TRUE, value := CONST.CUTTINGUNIT.CMDs.NO_CMD);
			busy := FALSE;
			state := ST_IDLE;
//		ELSIF config.busy OR config.cmd <> CONST.CUTTINGUNIT.CMDs.NO_CMD THEN
//			config(cmd := CONST.CUTTINGUNIT.CMDs.NO_CMD, axis := axis, status := status);
		ELSE
			config(cmd := cmdStatus.value, axis := axis, status := status);
			state := ST_MOVE;
		END_IF

	ST_MOVE:
		config ( axis := axis, status := status);
		IF cmdCtrl.value = CONST.CUTTINGUNIT.CMDs.NO_CMD THEN
			config(cmd := CONST.CUTTINGUNIT.CMDs.NO_CMD,  axis := axis, status := status);
			state := ST_MOVE_QUIT;
		END_IF

	ST_MOVE_QUIT:
		config(cmd := CONST.CUTTINGUNIT.CMDs.NO_CMD, axis := axis, status := status);
		IF NOT config.busy THEN
			busy := FALSE;
			unwinderOFF := FALSE;
			cmdStatus(set := TRUE, value := CONST.CUTTINGUNIT.CMDs.NO_CMD);
			state := ST_IDLE;
		END_IF

	ST_FUNCTION_START:
		IF config.busy OR config.cmd <> CONST.CUTTINGUNIT.CMDs.NO_CMD THEN
			config(cmd := CONST.CUTTINGUNIT.CMDs.NO_CMD, axis := axis, status := status);
		ELSE
			config(cmd := CONST.CUTTINGUNIT.CMDs.CALIBR (*cmdStatus.value*), axis := axis, status := status);
			state := ST_FUNCTION;
		END_IF

	ST_FUNCTION:
		config(  axis := axis, status := status);
		IF NOT config.busy THEN
			IF config.err.flag THEN
				err := config.err;
				err.state := state;
			END_IF
			config(cmd := CONST.CUTTINGUNIT.CMDs.NO_CMD,  axis := axis, status := status );
			state := ST_FUNCTION_QUIT;
		ELSIF keys.up.LDT.button AND keys.down.LDT.button THEN//10.11.15
				config(cmd := CONST.CUTTINGUNIT.CMDs.RESET,  axis := axis, status := status );
			state := ST_FUNCTION_QUIT;
		END_IF

	ST_FUNCTION_QUIT:
		busy := FALSE;

		IF cmdCtrl.value = CONST.CUTTINGUNIT.CMDs.NO_CMD THEN
			cmdStatus(set :=TRUE, value := CONST.CUTTINGUNIT.CMDs.NO_CMD);
			unwinderOFF := FALSE;
			state := ST_IDLE;
		END_IF

	END_CASE

END_ACTION
```

#### acSetModeAfterBuffer.st
```iecst
(********************************************************************
 * COPYRIGHT -- Microsoft
 ********************************************************************
 * Programm: MAIN
 * Datei: acSetModeAfterBuffer.st
 * Autor: awalz
 * Erstellt: 10. Juli 2014
 ********************************************************************
 * Implementierung des Programms MAIN
 ********************************************************************)

(* Fügt einae neue Aktion zum IEC Programm oder Bibliothek *)
ACTION acSetModeAfterBuffer:
	IF BetrCtrl.value = CONST.MACHINEMODES.EMERGENCYSTOP THEN
		StateCtrl := CTRL_EMERGENCYSTOP_BEFORE;
	ELSIF BetrCtrl.value = CONST.MACHINEMODES.SAFETYSTOP THEN
		StateCtrl := CTRL_SAFETYSTOP_BEFORE;
	ELSIF BetrCtrl.value = CONST.MACHINEMODES.MANUAL THEN
		StateCtrl := CTRL_STOP_BEFORE;
	ELSIF BetrCtrl.value = CONST.MACHINEMODES.AUTOMATIC THEN
		StateCtrl := CTRL_STOP_BEFORE;
	END_IF
END_ACTION
```

#### acBuffercyclic.st
```iecst
(********************************************************************
 * COPYRIGHT -- Microsoft
 ********************************************************************
 * Programm: MAIN
 * Datei: acBuffercyclic.st
 * Autor: awalz
 * Erstellt: 27. November 2014
 ********************************************************************
 * Implementierung des Programms MAIN
 ********************************************************************)

(* Fügt eine neue Aktion zum IEC Programm oder Bibliothek *)
ACTION acBuffercyclic:

	IF axis.ctrl.MC_ReadActualPosition_0.Position > 6555 AND axis.bufferaxis.MC_BR_VelocityControl_0.Active  THEN
		axis.bufferaxis.cmd := CONST.AXIS.STOP; (* da kein Endlageschalter vorhanden Moment abschalten*)
	END_IF

	IF keys.up.LDT.button THEN
			axis.bufferaxis.cmd := CONST.AXIS.JOG_POS;
	ELSIF keys.down.LDT.button THEN
			axis.bufferaxis.cmd := CONST.AXIS.JOG_NEG;
	ELSIF keys.down.LDT.ftrig.Q OR keys.up.LDT.ftrig.Q THEN
		axis.bufferaxis.cmd := CONST.AXIS.NOACTION;
//	ELSIF keys.home.LDT.button THEN
//		cmdCtrl.value := CONST.CUTTINGUNIT.CMDs.CALIBR;
//	ELSE
//		cmdCtrl.value := CONST.CUTTINGUNIT.CMDs.NO_CMD;
	END_IF
	buffertofullRtrig(CLK := online (*OR buffertofull*));

	IF NOT online THEN (*der Bahnspeicher darf nur bis zur Position X fahren*)
			axis.bufferaxis.override := 0;
		IF torquelow AND NOT keys.down.LDT.button AND NOT keys.up.LDT.button  THEN (*wird von der Klemmbalken gesetzt und soll der Speicher in Standstill versetzen*)
			axis.bufferaxis.cmd := CONST.AXIS.STOP;
		ELSIF axis.ctrl.MC_ReadActualPosition_0.Position > setposition 	AND  NOT keys.down.LDT.button AND NOT keys.up.LDT.button  THEN
			axis.bufferaxis.cmd := CONST.AXIS.STOP;
		ELSIF axis.ctrl.MC_ReadActualPosition_0.Position < setposition 	AND  NOT keys.down.LDT.button AND NOT keys.up.LDT.button AND NOT torquelow THEN
			axis.bufferaxis.cmd := CONST.AXIS.START;
		END_IF
	ELSE (*online muss der Puffer gefüllt werden bzw ständig voll sein*)
		IF torquelow THEN (*der Bahnspeicher darf bis zum oberen Endschalter fahren*)
			axis.bufferaxis.override := 0;
			axis.bufferaxis.cmd := CONST.AXIS.START;
		ELSE
			IF  axis.ctrl.MC_ReadActualPosition_0.Position < 6000 THEN (* Position gilt noch zu definieren*)
				axis.bufferaxis.override := 80; (* da beim Inlinebetrieb der Speicher keine Funktion hat*)
				axis.bufferaxis.cmd := CONST.AXIS.START;
			ELSIF  axis.ctrl.MC_ReadActualPosition_0.Position > 6000 THEN
				axis.bufferaxis.override := 0;
				axis.bufferaxis.cmd := CONST.AXIS.STOP;
			END_IF
		END_IF
	END_IF

END_ACTION
```
